IF VAR_mantisse2[2] >1 THEN
VAR_calcul_mantisse_temp.30:=TRUE;
VAR_mantisse2[2]:= VAR_mantisse2[2] -1;
ELSIF VAR_mantisse2[2] =1 THEN
VAR_calcul_mantisse_temp.30:=TRUE;
VAR_mantisse2[3]:=0;
VAR_mantisse2[4]:=0;
VAR_mantisse2[5]:=0;
VAR_mantisse2[6]:=0;
VAR_mantisse2[7]:=0;
VAR_mantisse2[8]:=0;
VAR_mantisse2[9]:=0;
VAR_mantisse2[10]:=0;
VAR_mantisse2[11]:=0;
VAR_mantisse2[12]:=0;
VAR_mantisse2[13]:=0;
VAR_mantisse2[14]:=0;
VAR_mantisse2[15]:=0;
VAR_mantisse2[16]:=0;
VAR_mantisse2[17]:=0;
VAR_mantisse2[18]:=0;
VAR_mantisse2[19]:=0;
VAR_mantisse2[20]:=0;
VAR_mantisse2[21]:=0;
VAR_mantisse2[22]:=0;
VAR_mantisse2[23]:=0;
VAR_mantisse2[24]:=0;
VAR_mantisse2[25]:=0;
VAR_mantisse2[26]:=0;
VAR_mantisse2[27]:=0;
VAR_mantisse2[28]:=0;
VAR_mantisse2[29]:=0;
VAR_mantisse2[30]:=0;
VAR_mantisse2[31]:=0;
VAR_mantisse2[32]:=0;
END_IF;

IF VAR_mantisse2[3] >1 THEN
VAR_calcul_mantisse_temp.29:=TRUE;
VAR_mantisse2[3]:= VAR_mantisse2[3] -1;
ELSIF VAR_mantisse2[3] =1 THEN
VAR_calcul_mantisse_temp.29:=TRUE;
VAR_mantisse2[4]:=0;
VAR_mantisse2[5]:=0;
VAR_mantisse2[6]:=0;
VAR_mantisse2[7]:=0;
VAR_mantisse2[8]:=0;
VAR_mantisse2[9]:=0;
VAR_mantisse2[10]:=0;
VAR_mantisse2[11]:=0;
VAR_mantisse2[12]:=0;
VAR_mantisse2[13]:=0;
VAR_mantisse2[14]:=0;
VAR_mantisse2[15]:=0;
VAR_mantisse2[16]:=0;
VAR_mantisse2[17]:=0;
VAR_mantisse2[18]:=0;
VAR_mantisse2[19]:=0;
VAR_mantisse2[20]:=0;
VAR_mantisse2[21]:=0;
VAR_mantisse2[22]:=0;
VAR_mantisse2[23]:=0;
VAR_mantisse2[24]:=0;
VAR_mantisse2[25]:=0;
VAR_mantisse2[26]:=0;
VAR_mantisse2[27]:=0;
VAR_mantisse2[28]:=0;
VAR_mantisse2[29]:=0;
VAR_mantisse2[30]:=0;
VAR_mantisse2[31]:=0;
VAR_mantisse2[32]:=0;
END_IF;

IF VAR_mantisse2[4] >1 THEN
VAR_calcul_mantisse_temp.28:=TRUE;
VAR_mantisse2[4]:= VAR_mantisse2[4] -1;
ELSIF VAR_mantisse2[4] =1 THEN
VAR_calcul_mantisse_temp.28:=TRUE;
VAR_mantisse2[5]:=0;
VAR_mantisse2[6]:=0;
VAR_mantisse2[7]:=0;
VAR_mantisse2[8]:=0;
VAR_mantisse2[9]:=0;
VAR_mantisse2[10]:=0;
VAR_mantisse2[11]:=0;
VAR_mantisse2[12]:=0;
VAR_mantisse2[13]:=0;
VAR_mantisse2[14]:=0;
VAR_mantisse2[15]:=0;
VAR_mantisse2[16]:=0;
VAR_mantisse2[17]:=0;
VAR_mantisse2[18]:=0;
VAR_mantisse2[19]:=0;
VAR_mantisse2[20]:=0;
VAR_mantisse2[21]:=0;
VAR_mantisse2[22]:=0;
VAR_mantisse2[23]:=0;
VAR_mantisse2[24]:=0;
VAR_mantisse2[25]:=0;
VAR_mantisse2[26]:=0;
VAR_mantisse2[27]:=0;
VAR_mantisse2[28]:=0;
VAR_mantisse2[29]:=0;
VAR_mantisse2[30]:=0;
VAR_mantisse2[31]:=0;
VAR_mantisse2[32]:=0;
END_IF;

IF VAR_mantisse2[5] >1 THEN
VAR_calcul_mantisse_temp.27:=TRUE;
VAR_mantisse2[5]:= VAR_mantisse2[5] -1;
ELSIF VAR_mantisse2[5] =1 THEN
VAR_calcul_mantisse_temp.27:=TRUE;
VAR_mantisse2[6]:=0;
VAR_mantisse2[7]:=0;
VAR_mantisse2[8]:=0;
VAR_mantisse2[9]:=0;
VAR_mantisse2[10]:=0;
VAR_mantisse2[11]:=0;
VAR_mantisse2[12]:=0;
VAR_mantisse2[13]:=0;
VAR_mantisse2[14]:=0;
VAR_mantisse2[15]:=0;
VAR_mantisse2[16]:=0;
VAR_mantisse2[17]:=0;
VAR_mantisse2[18]:=0;
VAR_mantisse2[19]:=0;
VAR_mantisse2[20]:=0;
VAR_mantisse2[21]:=0;
VAR_mantisse2[22]:=0;
VAR_mantisse2[23]:=0;
VAR_mantisse2[24]:=0;
VAR_mantisse2[25]:=0;
VAR_mantisse2[26]:=0;
VAR_mantisse2[27]:=0;
VAR_mantisse2[28]:=0;
VAR_mantisse2[29]:=0;
VAR_mantisse2[30]:=0;
VAR_mantisse2[31]:=0;
VAR_mantisse2[32]:=0;
END_IF;

IF VAR_mantisse2[6] >1 THEN
VAR_calcul_mantisse_temp.26:=TRUE;
VAR_mantisse2[6]:= VAR_mantisse2[6] -1;
ELSIF VAR_mantisse2[6] =1 THEN
VAR_calcul_mantisse_temp.26:=TRUE;
VAR_mantisse2[7]:=0;
VAR_mantisse2[8]:=0;
VAR_mantisse2[9]:=0;
VAR_mantisse2[10]:=0;
VAR_mantisse2[11]:=0;
VAR_mantisse2[12]:=0;
VAR_mantisse2[13]:=0;
VAR_mantisse2[14]:=0;
VAR_mantisse2[15]:=0;
VAR_mantisse2[16]:=0;
VAR_mantisse2[17]:=0;
VAR_mantisse2[18]:=0;
VAR_mantisse2[19]:=0;
VAR_mantisse2[20]:=0;
VAR_mantisse2[21]:=0;
VAR_mantisse2[22]:=0;
VAR_mantisse2[23]:=0;
VAR_mantisse2[24]:=0;
VAR_mantisse2[25]:=0;
VAR_mantisse2[26]:=0;
VAR_mantisse2[27]:=0;
VAR_mantisse2[28]:=0;
VAR_mantisse2[29]:=0;
VAR_mantisse2[30]:=0;
VAR_mantisse2[31]:=0;
VAR_mantisse2[32]:=0;
END_IF;

IF VAR_mantisse2[7] >1 THEN
VAR_calcul_mantisse_temp.25:=TRUE;
VAR_mantisse2[7]:= VAR_mantisse2[7] -1;
ELSIF VAR_mantisse2[7] =1 THEN
VAR_calcul_mantisse_temp.25:=TRUE;
VAR_mantisse2[8]:=0;
VAR_mantisse2[9]:=0;
VAR_mantisse2[10]:=0;
VAR_mantisse2[11]:=0;
VAR_mantisse2[12]:=0;
VAR_mantisse2[13]:=0;
VAR_mantisse2[14]:=0;
VAR_mantisse2[15]:=0;
VAR_mantisse2[16]:=0;
VAR_mantisse2[17]:=0;
VAR_mantisse2[18]:=0;
VAR_mantisse2[19]:=0;
VAR_mantisse2[20]:=0;
VAR_mantisse2[21]:=0;
VAR_mantisse2[22]:=0;
VAR_mantisse2[23]:=0;
VAR_mantisse2[24]:=0;
VAR_mantisse2[25]:=0;
VAR_mantisse2[26]:=0;
VAR_mantisse2[27]:=0;
VAR_mantisse2[28]:=0;
VAR_mantisse2[29]:=0;
VAR_mantisse2[30]:=0;
VAR_mantisse2[31]:=0;
VAR_mantisse2[32]:=0;
END_IF;

IF VAR_mantisse2[8] >1 THEN
VAR_calcul_mantisse_temp.24:=TRUE;
VAR_mantisse2[8]:= VAR_mantisse2[8] -1;
ELSIF VAR_mantisse2[8] =1 THEN
VAR_calcul_mantisse_temp.24:=TRUE;
VAR_mantisse2[9]:=0;
VAR_mantisse2[10]:=0;
VAR_mantisse2[11]:=0;
VAR_mantisse2[12]:=0;
VAR_mantisse2[13]:=0;
VAR_mantisse2[14]:=0;
VAR_mantisse2[15]:=0;
VAR_mantisse2[16]:=0;
VAR_mantisse2[17]:=0;
VAR_mantisse2[18]:=0;
VAR_mantisse2[19]:=0;
VAR_mantisse2[20]:=0;
VAR_mantisse2[21]:=0;
VAR_mantisse2[22]:=0;
VAR_mantisse2[23]:=0;
VAR_mantisse2[24]:=0;
VAR_mantisse2[25]:=0;
VAR_mantisse2[26]:=0;
VAR_mantisse2[27]:=0;
VAR_mantisse2[28]:=0;
VAR_mantisse2[29]:=0;
VAR_mantisse2[30]:=0;
VAR_mantisse2[31]:=0;
VAR_mantisse2[32]:=0;
END_IF;

IF VAR_mantisse2[9] >1 THEN
VAR_calcul_mantisse_temp.23:=TRUE;
VAR_mantisse2[9]:= VAR_mantisse2[9] -1;
ELSIF VAR_mantisse2[9] =1 THEN
VAR_calcul_mantisse_temp.23:=TRUE;
VAR_mantisse2[10]:=0;
VAR_mantisse2[11]:=0;
VAR_mantisse2[12]:=0;
VAR_mantisse2[13]:=0;
VAR_mantisse2[14]:=0;
VAR_mantisse2[15]:=0;
VAR_mantisse2[16]:=0;
VAR_mantisse2[17]:=0;
VAR_mantisse2[18]:=0;
VAR_mantisse2[19]:=0;
VAR_mantisse2[20]:=0;
VAR_mantisse2[21]:=0;
VAR_mantisse2[22]:=0;
VAR_mantisse2[23]:=0;
VAR_mantisse2[24]:=0;
VAR_mantisse2[25]:=0;
VAR_mantisse2[26]:=0;
VAR_mantisse2[27]:=0;
VAR_mantisse2[28]:=0;
VAR_mantisse2[29]:=0;
VAR_mantisse2[30]:=0;
VAR_mantisse2[31]:=0;
VAR_mantisse2[32]:=0;
END_IF;

IF VAR_mantisse2[10] >1 THEN
VAR_calcul_mantisse_temp.22:=TRUE;
VAR_mantisse2[10]:= VAR_mantisse2[10] -1;
ELSIF VAR_mantisse2[10] =1 THEN
VAR_calcul_mantisse_temp.22:=TRUE;
VAR_mantisse2[11]:=0;
VAR_mantisse2[12]:=0;
VAR_mantisse2[13]:=0;
VAR_mantisse2[14]:=0;
VAR_mantisse2[15]:=0;
VAR_mantisse2[16]:=0;
VAR_mantisse2[17]:=0;
VAR_mantisse2[18]:=0;
VAR_mantisse2[19]:=0;
VAR_mantisse2[20]:=0;
VAR_mantisse2[21]:=0;
VAR_mantisse2[22]:=0;
VAR_mantisse2[23]:=0;
VAR_mantisse2[24]:=0;
VAR_mantisse2[25]:=0;
VAR_mantisse2[26]:=0;
VAR_mantisse2[27]:=0;
VAR_mantisse2[28]:=0;
VAR_mantisse2[29]:=0;
VAR_mantisse2[30]:=0;
VAR_mantisse2[31]:=0;
VAR_mantisse2[32]:=0;
END_IF;
IF VAR_mantisse2[11] >1 THEN
VAR_calcul_mantisse_temp.21:=TRUE;
VAR_mantisse2[11]:= VAR_mantisse2[11] -1;
ELSIF VAR_mantisse2[11] =1 THEN
VAR_calcul_mantisse_temp.21:=TRUE;
VAR_mantisse2[12]:=0;
VAR_mantisse2[13]:=0;
VAR_mantisse2[14]:=0;
VAR_mantisse2[15]:=0;
VAR_mantisse2[16]:=0;
VAR_mantisse2[17]:=0;
VAR_mantisse2[18]:=0;
VAR_mantisse2[19]:=0;
VAR_mantisse2[20]:=0;
VAR_mantisse2[21]:=0;
VAR_mantisse2[22]:=0;
VAR_mantisse2[23]:=0;
VAR_mantisse2[24]:=0;
VAR_mantisse2[25]:=0;
VAR_mantisse2[26]:=0;
VAR_mantisse2[27]:=0;
VAR_mantisse2[28]:=0;
VAR_mantisse2[29]:=0;
VAR_mantisse2[30]:=0;
VAR_mantisse2[31]:=0;
VAR_mantisse2[32]:=0;
END_IF;
IF VAR_mantisse2[12] >1 THEN
VAR_calcul_mantisse_temp.20:=TRUE;
VAR_mantisse2[12]:= VAR_mantisse2[12] -1;
ELSIF VAR_mantisse2[12] =1 THEN
VAR_calcul_mantisse_temp.20:=TRUE;
VAR_mantisse2[13]:=0;
VAR_mantisse2[14]:=0;
VAR_mantisse2[15]:=0;
VAR_mantisse2[16]:=0;
VAR_mantisse2[17]:=0;
VAR_mantisse2[18]:=0;
VAR_mantisse2[19]:=0;
VAR_mantisse2[20]:=0;
VAR_mantisse2[21]:=0;
VAR_mantisse2[22]:=0;
VAR_mantisse2[23]:=0;
VAR_mantisse2[24]:=0;
VAR_mantisse2[25]:=0;
VAR_mantisse2[26]:=0;
VAR_mantisse2[27]:=0;
VAR_mantisse2[28]:=0;
VAR_mantisse2[29]:=0;
VAR_mantisse2[30]:=0;
VAR_mantisse2[31]:=0;
VAR_mantisse2[32]:=0;
END_IF;
IF VAR_mantisse2[13] >1 THEN
VAR_calcul_mantisse_temp.19:=TRUE;
VAR_mantisse2[13]:= VAR_mantisse2[13] -1;
ELSIF VAR_mantisse2[13] =1 THEN
VAR_calcul_mantisse_temp.19:=TRUE;
VAR_mantisse2[14]:=0;
VAR_mantisse2[15]:=0;
VAR_mantisse2[16]:=0;
VAR_mantisse2[17]:=0;
VAR_mantisse2[18]:=0;
VAR_mantisse2[19]:=0;
VAR_mantisse2[20]:=0;
VAR_mantisse2[21]:=0;
VAR_mantisse2[22]:=0;
VAR_mantisse2[23]:=0;
VAR_mantisse2[24]:=0;
VAR_mantisse2[25]:=0;
VAR_mantisse2[26]:=0;
VAR_mantisse2[27]:=0;
VAR_mantisse2[28]:=0;
VAR_mantisse2[29]:=0;
VAR_mantisse2[30]:=0;
VAR_mantisse2[31]:=0;
VAR_mantisse2[32]:=0;
END_IF;
IF VAR_mantisse2[14] >1 THEN
VAR_calcul_mantisse_temp.18:=TRUE;
VAR_mantisse2[14]:= VAR_mantisse2[14] -1;
ELSIF VAR_mantisse2[14] =1 THEN
VAR_calcul_mantisse_temp.18:=TRUE;
VAR_mantisse2[15]:=0;
VAR_mantisse2[16]:=0;
VAR_mantisse2[17]:=0;
VAR_mantisse2[18]:=0;
VAR_mantisse2[19]:=0;
VAR_mantisse2[20]:=0;
VAR_mantisse2[21]:=0;
VAR_mantisse2[22]:=0;
VAR_mantisse2[23]:=0;
VAR_mantisse2[24]:=0;
VAR_mantisse2[25]:=0;
VAR_mantisse2[26]:=0;
VAR_mantisse2[27]:=0;
VAR_mantisse2[28]:=0;
VAR_mantisse2[29]:=0;
VAR_mantisse2[30]:=0;
VAR_mantisse2[31]:=0;
VAR_mantisse2[32]:=0;
END_IF;

IF VAR_mantisse2[15] >1 THEN
VAR_calcul_mantisse_temp.17:=TRUE;
VAR_mantisse2[15]:= VAR_mantisse2[15] -1;
ELSIF VAR_mantisse2[15] =1 THEN
VAR_calcul_mantisse_temp.17:=TRUE;
VAR_mantisse2[16]:=0;
VAR_mantisse2[17]:=0;
VAR_mantisse2[18]:=0;
VAR_mantisse2[19]:=0;
VAR_mantisse2[20]:=0;
VAR_mantisse2[21]:=0;
VAR_mantisse2[22]:=0;
VAR_mantisse2[23]:=0;
VAR_mantisse2[24]:=0;
VAR_mantisse2[25]:=0;
VAR_mantisse2[26]:=0;
VAR_mantisse2[27]:=0;
VAR_mantisse2[28]:=0;
VAR_mantisse2[29]:=0;
VAR_mantisse2[30]:=0;
VAR_mantisse2[31]:=0;
VAR_mantisse2[32]:=0;
END_IF;
IF VAR_mantisse2[16] >1 THEN
VAR_calcul_mantisse_temp.16:=TRUE;
VAR_mantisse2[16]:= VAR_mantisse2[16] -1;
ELSIF VAR_mantisse2[16] =1 THEN
VAR_calcul_mantisse_temp.16:=TRUE;
VAR_mantisse2[17]:=0;
VAR_mantisse2[18]:=0;
VAR_mantisse2[19]:=0;
VAR_mantisse2[20]:=0;
VAR_mantisse2[21]:=0;
VAR_mantisse2[22]:=0;
VAR_mantisse2[23]:=0;
VAR_mantisse2[24]:=0;
VAR_mantisse2[25]:=0;
VAR_mantisse2[26]:=0;
VAR_mantisse2[27]:=0;
VAR_mantisse2[28]:=0;
VAR_mantisse2[29]:=0;
VAR_mantisse2[30]:=0;
VAR_mantisse2[31]:=0;
VAR_mantisse2[32]:=0;
END_IF;
IF VAR_mantisse2[17] >1 THEN
VAR_calcul_mantisse_temp.15:=TRUE;
VAR_mantisse2[17]:= VAR_mantisse2[17] -1;
ELSIF VAR_mantisse2[17] =1 THEN
VAR_calcul_mantisse_temp.15:=TRUE;
VAR_mantisse2[18]:=0;
VAR_mantisse2[19]:=0;
VAR_mantisse2[20]:=0;
VAR_mantisse2[21]:=0;
VAR_mantisse2[22]:=0;
VAR_mantisse2[23]:=0;
VAR_mantisse2[24]:=0;
VAR_mantisse2[25]:=0;
VAR_mantisse2[26]:=0;
VAR_mantisse2[27]:=0;
VAR_mantisse2[28]:=0;
VAR_mantisse2[29]:=0;
VAR_mantisse2[30]:=0;
VAR_mantisse2[31]:=0;
VAR_mantisse2[32]:=0;
END_IF;
IF VAR_mantisse2[18] >1 THEN
VAR_calcul_mantisse_temp.14:=TRUE;
VAR_mantisse2[18]:= VAR_mantisse2[18] -1;
ELSIF VAR_mantisse2[18] =1 THEN
VAR_calcul_mantisse_temp.14:=TRUE;
VAR_mantisse2[19]:=0;
VAR_mantisse2[20]:=0;
VAR_mantisse2[21]:=0;
VAR_mantisse2[22]:=0;
VAR_mantisse2[23]:=0;
VAR_mantisse2[24]:=0;
VAR_mantisse2[25]:=0;
VAR_mantisse2[26]:=0;
VAR_mantisse2[27]:=0;
VAR_mantisse2[28]:=0;
VAR_mantisse2[29]:=0;
VAR_mantisse2[30]:=0;
VAR_mantisse2[31]:=0;
VAR_mantisse2[32]:=0;
END_IF;
IF VAR_mantisse2[19] >1 THEN
VAR_calcul_mantisse_temp.13:=TRUE;
VAR_mantisse2[19]:= VAR_mantisse2[19] -1;
ELSIF VAR_mantisse2[19] =1 THEN
VAR_calcul_mantisse_temp.13:=TRUE;
VAR_mantisse2[20]:=0;
VAR_mantisse2[21]:=0;
VAR_mantisse2[22]:=0;
VAR_mantisse2[23]:=0;
VAR_mantisse2[24]:=0;
VAR_mantisse2[25]:=0;
VAR_mantisse2[26]:=0;
VAR_mantisse2[27]:=0;
VAR_mantisse2[28]:=0;
VAR_mantisse2[29]:=0;
VAR_mantisse2[30]:=0;
VAR_mantisse2[31]:=0;
VAR_mantisse2[32]:=0;
END_IF;
IF VAR_mantisse2[20] >1 THEN
VAR_calcul_mantisse_temp.12:=TRUE;
VAR_mantisse2[20]:= VAR_mantisse2[20] -1;
ELSIF VAR_mantisse2[20] =1 THEN
VAR_calcul_mantisse_temp.12:=TRUE;
VAR_mantisse2[21]:=0;
VAR_mantisse2[22]:=0;
VAR_mantisse2[23]:=0;
VAR_mantisse2[24]:=0;
VAR_mantisse2[25]:=0;
VAR_mantisse2[26]:=0;
VAR_mantisse2[27]:=0;
VAR_mantisse2[28]:=0;
VAR_mantisse2[29]:=0;
VAR_mantisse2[30]:=0;
VAR_mantisse2[31]:=0;
VAR_mantisse2[32]:=0;
END_IF;
IF VAR_mantisse2[21] >1 THEN
VAR_calcul_mantisse_temp.11:=TRUE;
VAR_mantisse2[21]:= VAR_mantisse2[21] -1;
ELSIF VAR_mantisse2[21] =1 THEN
VAR_calcul_mantisse_temp.11:=TRUE;
VAR_mantisse2[22]:=0;
VAR_mantisse2[23]:=0;
VAR_mantisse2[24]:=0;
VAR_mantisse2[25]:=0;
VAR_mantisse2[26]:=0;
VAR_mantisse2[27]:=0;
VAR_mantisse2[28]:=0;
VAR_mantisse2[29]:=0;
VAR_mantisse2[30]:=0;
VAR_mantisse2[31]:=0;
VAR_mantisse2[32]:=0;
END_IF;
IF VAR_mantisse2[22] >1 THEN
VAR_calcul_mantisse_temp.10:=TRUE;
VAR_mantisse2[22]:= VAR_mantisse2[22] -1;
ELSIF VAR_mantisse2[22] =1 THEN
VAR_calcul_mantisse_temp.10:=TRUE;
VAR_mantisse2[23]:=0;
VAR_mantisse2[24]:=0;
VAR_mantisse2[25]:=0;
VAR_mantisse2[26]:=0;
VAR_mantisse2[27]:=0;
VAR_mantisse2[28]:=0;
VAR_mantisse2[29]:=0;
VAR_mantisse2[30]:=0;
VAR_mantisse2[31]:=0;
VAR_mantisse2[32]:=0;
END_IF;
IF VAR_mantisse2[23] >1 THEN
VAR_calcul_mantisse_temp.9:=TRUE;
VAR_mantisse2[23]:= VAR_mantisse2[23] -1;
ELSIF VAR_mantisse2[23] =1 THEN
VAR_calcul_mantisse_temp.9:=TRUE;
VAR_mantisse2[24]:=0;
VAR_mantisse2[25]:=0;
VAR_mantisse2[26]:=0;
VAR_mantisse2[27]:=0;
VAR_mantisse2[28]:=0;
VAR_mantisse2[29]:=0;
VAR_mantisse2[30]:=0;
VAR_mantisse2[31]:=0;
VAR_mantisse2[32]:=0;
END_IF;
IF VAR_mantisse2[24] >1 THEN
VAR_calcul_mantisse_temp.8:=TRUE;
VAR_mantisse2[24]:= VAR_mantisse2[24] -1;
ELSIF VAR_mantisse2[24] =1 THEN
VAR_calcul_mantisse_temp.8:=TRUE;
VAR_mantisse2[25]:=0;
VAR_mantisse2[26]:=0;
VAR_mantisse2[27]:=0;
VAR_mantisse2[28]:=0;
VAR_mantisse2[29]:=0;
VAR_mantisse2[30]:=0;
VAR_mantisse2[31]:=0;
VAR_mantisse2[32]:=0;
END_IF;
IF VAR_mantisse2[25] >1 THEN
VAR_calcul_mantisse_temp.7:=TRUE;
VAR_mantisse2[25]:= VAR_mantisse2[25] -1;
ELSIF VAR_mantisse2[25] =1 THEN
VAR_calcul_mantisse_temp.7:=TRUE;
VAR_mantisse2[26]:=0;
VAR_mantisse2[27]:=0;
VAR_mantisse2[28]:=0;
VAR_mantisse2[29]:=0;
VAR_mantisse2[30]:=0;
VAR_mantisse2[31]:=0;
VAR_mantisse2[32]:=0;
END_IF;
IF VAR_mantisse2[26] >1 THEN
VAR_calcul_mantisse_temp.6:=TRUE;
VAR_mantisse2[26]:= VAR_mantisse2[26] -1;
ELSIF VAR_mantisse2[26] =1 THEN
VAR_calcul_mantisse_temp.6:=TRUE;
VAR_mantisse2[27]:=0;
VAR_mantisse2[28]:=0;
VAR_mantisse2[29]:=0;
VAR_mantisse2[30]:=0;
VAR_mantisse2[31]:=0;
VAR_mantisse2[32]:=0;
END_IF;
IF VAR_mantisse2[27] >1 THEN
VAR_calcul_mantisse_temp.5:=TRUE;
VAR_mantisse2[27]:= VAR_mantisse2[27] -1;
ELSIF VAR_mantisse2[27] =1 THEN
VAR_calcul_mantisse_temp.5:=TRUE;
VAR_mantisse2[28]:=0;
VAR_mantisse2[29]:=0;
VAR_mantisse2[30]:=0;
VAR_mantisse2[31]:=0;
VAR_mantisse2[32]:=0;
END_IF;
IF VAR_mantisse2[28] >1 THEN
VAR_calcul_mantisse_temp.4:=TRUE;
VAR_mantisse2[28]:= VAR_mantisse2[28] -1;
ELSIF VAR_mantisse2[28] =1 THEN
VAR_calcul_mantisse_temp.4:=TRUE;
VAR_mantisse2[29]:=0;
VAR_mantisse2[30]:=0;
VAR_mantisse2[31]:=0;
VAR_mantisse2[32]:=0;
END_IF;
IF VAR_mantisse2[29] >1 THEN
VAR_calcul_mantisse_temp.3:=TRUE;
VAR_mantisse2[29]:= VAR_mantisse2[29] -1;
ELSIF VAR_mantisse2[29] =1 THEN
VAR_calcul_mantisse_temp.3:=TRUE;
VAR_mantisse2[30]:=0;
VAR_mantisse2[31]:=0;
VAR_mantisse2[32]:=0;
END_IF;
IF VAR_mantisse2[30] >1 THEN
VAR_calcul_mantisse_temp.2:=TRUE;
VAR_mantisse2[30]:= VAR_mantisse2[30] -1;
ELSIF VAR_mantisse2[30] =1 THEN
VAR_calcul_mantisse_temp.2:=TRUE;
VAR_mantisse2[31]:=0;
VAR_mantisse2[32]:=0;
END_IF;
IF VAR_mantisse2[31] >1 THEN
VAR_calcul_mantisse_temp.1:=TRUE;
VAR_mantisse2[31]:= VAR_mantisse2[31] -1;
ELSIF VAR_mantisse2[31] =1 THEN
VAR_calcul_mantisse_temp.1:=TRUE;
VAR_mantisse2[32]:=0;
END_IF;
IF VAR_mantisse2[32] >1 THEN
VAR_calcul_mantisse_temp.0:=TRUE;
VAR_mantisse2[32]:= VAR_mantisse2[32] -1;
ELSIF VAR_mantisse2[32] =1 THEN
VAR_calcul_mantisse_temp.0:=TRUE;
END_IF;
END_FOR

VAR_calcul_mantisse_temp2:=VAR_calcul_mantisse_temp;
VAR_value2:=VAR_value_entiere_corrige;
N:=0;
FOR I:=1 TO 32 DO

IF VAR_mantisse2[I] = 1 THEN
	N:=INT_TO_BYTE(I);
END_IF
END_FOR

Var_decalage_bit:=32-N;
VAR_mantisse_decimal:=ROR(VAR_calcul_mantisse_temp2,Var_decalage_bit);
VAR_mantisse_entier:=ROL(VAR_value2,N);

VAR_mantisse_final:= VAR_mantisse_entier OR VAR_mantisse_decimal;

IF VAR_mantisse_final.31=TRUE THEN
VAR_nb_zero:=0;
ELSIF VAR_mantisse_final.30=TRUE THEN
VAR_nb_zero:=1;
ELSIF VAR_mantisse_final.29=TRUE THEN
VAR_nb_zero:=2;
ELSIF VAR_mantisse_final.28=TRUE THEN
VAR_nb_zero:=3;
ELSIF VAR_mantisse_final.27=TRUE THEN
VAR_nb_zero:=4;
ELSIF VAR_mantisse_final.26=TRUE THEN
VAR_nb_zero:=5;
ELSIF VAR_mantisse_final.25=TRUE THEN
VAR_nb_zero:=6;
ELSIF VAR_mantisse_final.24=TRUE THEN
VAR_nb_zero:=7;
ELSIF VAR_mantisse_final.23=TRUE THEN
VAR_nb_zero:=8;
ELSIF VAR_mantisse_final.22=TRUE THEN
VAR_nb_zero:=9;
ELSIF VAR_mantisse_final.21=TRUE THEN
VAR_nb_zero:=10;
ELSIF VAR_mantisse_final.20=TRUE THEN
VAR_nb_zero:=11;
ELSIF VAR_mantisse_final.19=TRUE THEN
VAR_nb_zero:=12;
ELSIF VAR_mantisse_final.18=TRUE THEN
VAR_nb_zero:=13;
ELSIF VAR_mantisse_final.17=TRUE THEN
VAR_nb_zero:=14;
ELSIF VAR_mantisse_final.16=TRUE THEN
VAR_nb_zero:=15;
ELSIF VAR_mantisse_final.15=TRUE THEN
VAR_nb_zero:=16;
ELSIF VAR_mantisse_final.14=TRUE THEN
VAR_nb_zero:=17;
ELSIF VAR_mantisse_final.13=TRUE THEN
VAR_nb_zero:=18;
ELSIF VAR_mantisse_final.12=TRUE THEN
VAR_nb_zero:=19;
ELSIF VAR_mantisse_final.11=TRUE THEN
VAR_nb_zero:=20;
ELSIF VAR_mantisse_final.10=TRUE THEN
VAR_nb_zero:=21;
ELSIF VAR_mantisse_final.9=TRUE THEN
VAR_nb_zero:=22;
ELSIF VAR_mantisse_final.8=TRUE THEN
VAR_nb_zero:=23;
ELSIF VAR_mantisse_final.7=TRUE THEN
VAR_nb_zero:=24;
ELSIF VAR_mantisse_final.6=TRUE THEN
VAR_nb_zero:=25;
ELSIF VAR_mantisse_final.5=TRUE THEN
VAR_nb_zero:=26;
ELSIF VAR_mantisse_final.4=TRUE THEN
VAR_nb_zero:=27;
ELSIF VAR_mantisse_final.3=TRUE THEN
VAR_nb_zero:=28;
ELSIF VAR_mantisse_final.2=TRUE THEN
VAR_nb_zero:=29;
ELSIF VAR_mantisse_final.1=TRUE THEN
VAR_nb_zero:=30;
ELSIF VAR_mantisse_final.0=TRUE THEN
VAR_nb_zero:=31;
END_IF

 VAR_calcul_exposant := (32 - VAR_nb_zero - N - 1) + 127;

J:=INT_TO_BYTE(VAR_nb_zero);

VAR_mantisse_final2:=ROL(VAR_mantisse_final ,J);

VAR_calcul_sortie.31 := VAR_signe;

VAR_calcul_sortie.30 := VAR_calcul_exposant.7;
VAR_calcul_sortie.29 := VAR_calcul_exposant.6;
VAR_calcul_sortie.28 := VAR_calcul_exposant.5;
VAR_calcul_sortie.27 := VAR_calcul_exposant.4 ;
VAR_calcul_sortie.26 := VAR_calcul_exposant.3;
VAR_calcul_sortie.25 := VAR_calcul_exposant.2;
VAR_calcul_sortie.24 := VAR_calcul_exposant.1 ;
VAR_calcul_sortie.23 := VAR_calcul_exposant.0;

VAR_calcul_sortie.22 := VAR_mantisse_final2.30;
VAR_calcul_sortie.21 := VAR_mantisse_final2.29;
VAR_calcul_sortie.20 := VAR_mantisse_final2.28;
VAR_calcul_sortie.19 := VAR_mantisse_final2.27;
VAR_calcul_sortie.18 := VAR_mantisse_final2.26;
VAR_calcul_sortie.17 := VAR_mantisse_final2.25;
VAR_calcul_sortie.16 := VAR_mantisse_final2.24;
VAR_calcul_sortie.15 := VAR_mantisse_final2.23;
VAR_calcul_sortie.14 := VAR_mantisse_final2.22;
VAR_calcul_sortie.13 := VAR_mantisse_final2.21;
VAR_calcul_sortie.12 := VAR_mantisse_final2.20;
VAR_calcul_sortie.11 := VAR_mantisse_final2.19;
VAR_calcul_sortie.10 := VAR_mantisse_final2.18;
VAR_calcul_sortie.9 := VAR_mantisse_final2.17;
VAR_calcul_sortie.8 := VAR_mantisse_final2.16;
VAR_calcul_sortie.7 := VAR_mantisse_final2.15;
VAR_calcul_sortie.6 := VAR_mantisse_final2.14;
VAR_calcul_sortie.5 := VAR_mantisse_final2.13;
VAR_calcul_sortie.4 := VAR_mantisse_final2.12;
VAR_calcul_sortie.3 := VAR_mantisse_final2.11;
VAR_calcul_sortie.2 := VAR_mantisse_final2.10;
VAR_calcul_sortie.1 := VAR_mantisse_final2.9;
VAR_calcul_sortie.0 := VAR_mantisse_final2.8;

OUTPUT[0].0 := VAR_calcul_sortie.0;
OUTPUT[0].1 := VAR_calcul_sortie.1;
OUTPUT[0].2 := VAR_calcul_sortie.2;
OUTPUT[0].3 := VAR_calcul_sortie.3;
OUTPUT[0].4 := VAR_calcul_sortie.4;
OUTPUT[0].5 := VAR_calcul_sortie.5;
OUTPUT[0].6 := VAR_calcul_sortie.6;
OUTPUT[0].7 := VAR_calcul_sortie.7;

OUTPUT[1].0 := VAR_calcul_sortie.8;
OUTPUT[1].1 := VAR_calcul_sortie.9;
OUTPUT[1].2 := VAR_calcul_sortie.10;
OUTPUT[1].3 := VAR_calcul_sortie.11;
OUTPUT[1].4 := VAR_calcul_sortie.12;
OUTPUT[1].5 := VAR_calcul_sortie.13;
OUTPUT[1].6 := VAR_calcul_sortie.14;
OUTPUT[1].7 := VAR_calcul_sortie.15;

OUTPUT[2].0 := VAR_calcul_sortie.16;
OUTPUT[2].1 := VAR_calcul_sortie.17;
OUTPUT[2].2 := VAR_calcul_sortie.18;
OUTPUT[2].3 := VAR_calcul_sortie.19;
OUTPUT[2].4 := VAR_calcul_sortie.20;
OUTPUT[2].5 := VAR_calcul_sortie.21;
OUTPUT[2].6 := VAR_calcul_sortie.22;
OUTPUT[2].7 := VAR_calcul_sortie.23;

OUTPUT[3].0 := VAR_calcul_sortie.24;
OUTPUT[3].1 := VAR_calcul_sortie.25;
OUTPUT[3].2 := VAR_calcul_sortie.26;
OUTPUT[3].3 := VAR_calcul_sortie.27;
OUTPUT[3].4 := VAR_calcul_sortie.28;
OUTPUT[3].5 := VAR_calcul_sortie.29;
OUTPUT[3].6 := VAR_calcul_sortie.30;
OUTPUT[3].7 := VAR_calcul_sortie.31;

END_FUNCTION_BLOCK

// ---- POUs/Fonction/ETHER COM/BLOCK_XTC_CLIENT_EXCHANGE.TcPOU
FUNCTION_BLOCK BLOCK_XTC_CLIENT_EXCHANGE
(* Fonction de lecture / écriture sur port TcpIP*)
(* version 0 - SP - 24/02/2015*)


VAR_INPUT
	hSocket				: T_HSOCKET;	(*socket*)
	TxBuffer				: ARRAY[0..MAX_TXBUFFER_SIZE] OF BYTE;
	bExecute			: BOOL;			(*bit de déclenchelent de l'émission/réception - sur front montant*)
	nbExpectedChar		: UDINT;			(*nombre de caractère attendu en réception*)
	nbTransmittedChar	: UDINT;			(*nombre de caractère transmis à l'émission*)
	PRM_RECEIVE_POLLING_TIME		 		: TIME := T#1s;	(*temporisation de polling de réception*)
	PRM_RECEIVE_TIMEOUT						: TIME := T#10s;	(*temporisation de timeout de communication*)

END_VAR
VAR_OUTPUT
	bBusy 				: BOOL;			(*processus d'emission/réception occupé*)
	bError				: BOOL;			(*processus d'emission/réception en erreur*)
	nErrId				: UDINT;			(*n° d'erreur*)
	nstepInError			: UDINT;			(*n° d'étape sur laquelle s'est produite l'erreur*)
	ErrDescription		: T_MaxString;	(*chaine de caractère d'intitulé de l'erreur*)
	rxBuffer				: ARRAY[0..MAX_RXBUFFER_SIZE] OF BYTE; (*réponse du serveur en mode buffer*)
	STATE_Com_Err_Counter:	UDINT;
	STATE_nbReceptedChar:	UDINT;			(*nombre effectif de caractère recu - peut différer du nombre de caractère attendu dans le cas d'une trame
										d'erreur*)

END_VAR
VAR
	fbSocketSend		: FB_SocketSend := ( sSrvNetID := '', tTimeout := DEFAULT_ADS_TIMEOUT );
	fbSocketReceive		: FB_SocketReceive := ( sSrvNetID := '', tTimeout := DEFAULT_ADS_TIMEOUT );
	fbReceiveTON		: TON;		(*tempo pour polling de réception*)
	fbDisconnectTON		: TON;		(*tempo de time out*)
	RisingEdge			: R_TRIG;
	eStep				: E_DataExchaSteps;
	cbReceived, startPos, endPos, idx	: UDINT;
	cbFrame				: UDINT;
	Temp_rxBuffer		: ARRAY[0..MAX_RXBUFFER_SIZE] OF BYTE;
	I					: INT; 		(*Compteur d'itération*)
	LOG_COM			: ARRAY[0..MAX_BUFFER_DIALOG] OF STRUCT_LOG_TCPIP_CLIENT;	(*buffer de chaine en émission*)
	VAR_COUNT_RETRY:	INT;		(*Compteur de tentative de retransmission du paramètre*)
END_VAR
VAR_TEMP
	Temp_byte:			BYTE;
END_VAR

RisingEdge( CLK := bExecute );	(*gestion du front montant de la demande d'exécution*)
CASE eStep OF

	DATAEXCHA_STATE_IDLE:	(*etape 0 - fonction d'émisson réception à l'arrêt*)
		IF RisingEdge.Q THEN		(*demande d'emission/réception sur FM du bit bexecute*)
		VAR_COUNT_RETRY := 0;
			(*RAZ du buffer de réception et du buffer de réception temporaire*)
			FOR i:=0 TO UDINT_TO_INT(MAX_RXBUFFER_SIZE) DO
				Temp_RxBuffer[i] := 0;
				RxBuffer[i] :=0;
			END_FOR
			bBusy := TRUE;							(*processus d'émission / réception occupé*)
			bError := FALSE;							(* RAZ drapeau d'erreur*)
			nErrid := 0;								(*RAZ du type d'érreur*)
			fbReceiveTON( IN := FALSE, PT := T#0s ); 	(* Réglage du buffer de réception à 0 pour lire asap *)
			fbDisconnectTON( IN := FALSE, PT := T#0s );	(* désactivation du timer de timeout *)
			eStep := DATAEXCHA_STATE_SEND_START;
		END_IF

	DATAEXCHA_STATE_SEND_START:		(*Etape 1 -  Envoi de la trame au serveur*)
		fbSocketSend( bExecute := FALSE );
		CbReceived := 0;
		(*on envoie le buffer d'émission*)
		fbSocketSend(
					hSocket	:= hSocket,
					pSrc	:= ADR(TxBuffer),
					cblen 	:= NbTransmittedChar, (* longueur de chaine sans le délimiteur *)
					bExecute:= TRUE,
					);
		fbsocketSend.cblen := NbTransmittedChar; (*longueur de chaine à envoyer*)

		SHIFT_BUFFER_DIALOG(); (*décalage du buffer de mémoire des dernières trames d'émission*)

		(*mémorisation du buffer d'émission dans le journal des échanges *)
		 MEMCPY( ADR(LOG_COM[0].TX),ADR(TxBuffer),FbSocketSend.Cblen);

		eStep := DATAEXCHA_STATE_SEND_WAIT;

	DATAEXCHA_STATE_SEND_WAIT:			(* Etape 2 - attente de la fin de l'envoi de la trame*)
		fbSocketSend( bExecute := FALSE );
		IF NOT fbSocketSend.bBusy THEN	(*si fin de l'emission*)
			IF NOT fbSocketSend.bError THEN	(*pas d'erreur*)
				eStep := DATAEXCHA_STATE_RECEIVE_START;
			ELSE	(*detection d'une erreur d'émission*)
				(*LogError( 'FB_SocketSend (local client)', fbSocketSend.nErrId );*)
				nErrId := fbSocketSend.nErrId;
				nstepInError := 2;
				ErrDescription := CONCAT('FB_ClientDataExcha - SENDING ERROR: ', UDINT_TO_STRING(nErrId));
				LOG_COM[0].ERR := ErrDescription;
				eStep := DATAEXCHA_STATE_ERROR;
			END_IF
		END_IF

	DATAEXCHA_STATE_RECEIVE_START: 	(*Etape 3 - gestion de la réception*)
		fbDisconnectTON(  );	(*lancement de la tempo de timeout : desactivée au premier appel*)
		fbReceiveTON( IN := TRUE );	(*temporisation de polling de reception - lancé avec délai 0ms au premier appel*)
		IF fbReceiveTON.Q THEN
			fbReceiveTON( IN := FALSE );
			fbSocketReceive( bExecute := FALSE );
			fbSocketReceive(  hSocket:= hSocket,
							pDest:= ADR( Temp_rxBuffer ) + cbReceived,	(*ajouté au buffer de réception à partir du dernier index CbReceived*)
							cbLen:= SIZEOF( Temp_rxBuffer ) - cbReceived,   (*longueur max = longeur du buffer - dernier index CbReceived*)
							bExecute:= TRUE );
			eStep := DATAEXCHA_STATE_RECEIVE_WAIT;
		END_IF

	DATAEXCHA_STATE_RECEIVE_WAIT:			(*étape 4 - attente de la fin de réception*)
		fbSocketReceive( bExecute := FALSE );
		IF NOT fbSocketReceive.bBusy THEN		(*si pas fonction de réception en cours*)
			IF NOT fbSocketReceive.bError THEN	(*si pas d'erreur*)
				(*et si des bytes ont été reçu*)
				IF (fbSocketReceive.nRecBytes > 0) THEN(* si on a reçu des informations *)
					startPos 		:= cbReceived;(* calcul de l'index de début de la nouvelle trame lue dans le buffer *)
					endPos  		:= cbReceived + fbSocketReceive.nRecBytes  - 1;(* calcul de l'index de fin de la nouvelle trame lue dans le buffer *)
					cbReceived 	:= cbReceived + fbSocketReceive.nRecBytes;(* recalcule le nombre total de caractères reçus depuis la requête en émission*)
					cbFrame		:= 0;(* remise à 0 de la  *)

					IF  (cbReceived < MAX_RXBUFFER_SIZE) (* contrôle de débordement *)  THEN

						fbReceiveTON( PT := T#0s ); (* bytes reçus =>on fixe la pariode de pooling a 0ms *)
						fbDisconnectTON( IN := FALSE );(* bytes recus => on ihnibe la tempo de timeout *)

						(*analyse des 2 premiers octets de la trame*)
						IF (cbReceived >=3)  THEN
							(*reception d'un message d'erreur de l'XTC*)
							IF ((temp_RxBuffer[0] + (Temp_RxBuffer[1] * 256)) = 6) AND (Temp_RxBuffer[2] = 16#80) THEN
								nbExpectedChar:= 6;	(*on corrige le nombre de caractère attendu*)
								STATE_nbReceptedChar:=6;
							END_IF
							(*Reception d'un message au format erroné - mauvais caractère CCB*)
							IF NOT (Temp_RxBuffer[2] = 16#00) AND NOT (Temp_RxBuffer[2] = 16#80) THEN
								STATE_nbReceptedChar:=(temp_RxBuffer[0] + (Temp_RxBuffer[1] * 256)) + 3;
								nErrId := ERROR_MESSAGE_CCB;	(*CCB incohérent*)
								nstepInError := 4;
								ErrDescription := 'FB_ClientDataExcha - Bad CCB';
								LOG_COM[0].ERR := ErrDescription;
								MEMCPY( ADR(LOG_COM[0].RX),ADR(Temp_RxBuffer),MAX_RXBUFFER_SIZE+1);	(*enregistrement dans le journal d'échange*)
								eStep := DATAEXCHA_STATE_ERROR;
							(*la longeur effective de la trame donnée par le premier octet  n'est pas cohérente avec la longueur attendue*)
							(*alors erreur*)
							ELSIF NOT ((temp_RxBuffer[0] + (Temp_RxBuffer[1] * 256) + 3) = NbExpectedChar) THEN
								STATE_nbReceptedChar:=(temp_RxBuffer[0] + (Temp_RxBuffer[1] * 256)) + 3;
								nErrId := ERROR_MESSAGE_LENGTH;	(*longueur trame incoérente*)
								nstepInError := 4;
								ErrDescription := 'FB_ClientDataExcha - Bad message length';
								LOG_COM[0].ERR := ErrDescription;
								MEMCPY( ADR(LOG_COM[0].RX),ADR(Temp_RxBuffer),MAX_RXBUFFER_SIZE+1);	(*enregistrement dans le journal d'échange*)
								eStep := DATAEXCHA_STATE_ERROR;
							ELSIF  (CbReceived >= nbExpectedChar) THEN	(*si le nombre de caractère reçu >= au nombre de caractère attendu*)
								(*Verification que la chaine recue comporte bien un caractère d'acquittement si le CCB = 0*)
								STATE_nbReceptedChar:=nbExpectedChar;
								IF NOT (Temp_RxBuffer[4] = 16#06) AND (Temp_RxBuffer[2] = 16#00) THEN
									STATE_nbReceptedChar:=(temp_RxBuffer[0] + (Temp_RxBuffer[1] * 256)) + 3;
									nErrId := ERROR_MISSING_ACK;	(*longueur trame incohérente*)
									nstepInError := 4;
									ErrDescription := 'FB_ClientDataExcha - Missing ACK';
									LOG_COM[0].ERR := ErrDescription;
									MEMCPY( ADR(LOG_COM[0].RX),ADR(Temp_RxBuffer),MAX_RXBUFFER_SIZE+1);	(*enregistrement dans le journal d'échange*)
									eStep := DATAEXCHA_STATE_ERROR;
								ELSE
									(*Calcul du CRC theorique*)
									Temp_Byte := 0;
										FOR I:=2 TO UDINT_TO_INT(nbExpectedChar-2) DO
											Temp_byte := Temp_Byte + Temp_RxBuffer[I];
										END_FOR
									(*si le CRC theorique n'est pas égal au CRC effectif alors erreur*)
									IF NOT (Temp_byte = temp_RxBuffer[NbExpectedChar-1])THEN
										STATE_nbReceptedChar:=(temp_RxBuffer[0] + (Temp_RxBuffer[1] * 256)) + 3;
										nErrId := ERROR_MESSAGE_LENGTH;	(*longueur trame incoérente*)
										nstepInError := 4;
										ErrDescription := 'FB_ClientDataExcha - Bad CRC';
										LOG_COM[0].ERR := ErrDescription;
										MEMCPY( ADR(LOG_COM[0].RX),ADR(Temp_RxBuffer),MAX_RXBUFFER_SIZE+1);	(*enregistrement dans le journal d'échange*)
										eStep := DATAEXCHA_STATE_ERROR;
										(*Tout est ok - on copy le buffer de réception temporaire dans le buffer de reception définitif*)
									ELSE
										MEMCPY(  ADR( RxBuffer ), ADR( Temp_rxBuffer ), NbExpectedChar); (*on récupère la chaine dans le buffer*)
										bBusy := FALSE;						(*Raz de l'indicateur de fonction d'émission/réception en cours*)
										VAR_COUNT_RETRY := 0; 				(*Raz du compteur de tentative de communication*)
										NErrId := 0;
										ErrDescription := 'NO ERROR ';
										nstepInError := 0;
										STATE_nbReceptedChar:=(temp_RxBuffer[0] + (Temp_RxBuffer[1] * 256)) + 3;
										eStep := DATAEXCHA_STATE_IDLE;
										LOG_COM[0].ERR := 'OK';
								 		MEMCPY( ADR(LOG_COM[0].RX),ADR(Temp_RxBuffer),NbExpectedChar);
									END_IF
								END_IF
							ELSE
								eStep := DATAEXCHA_STATE_RECEIVE_START; (* on répète l'étape de reception *)
							END_IF
						END_IF
					ELSE (* si il n'y a plus d'espace dispo dans le buffer *)
						nErrId := ERROR_RECEIVE_BUFFER_OVERFLOW;	(* buffer overflow !*)
						nstepInError := 4;
						ErrDescription := 'FB_ClientDataExcha - BUFFER OVERFLOW';
						LOG_COM[0].ERR := ErrDescription;
						MEMCPY( ADR(LOG_COM[0].RX),ADR(Temp_RxBuffer),MAX_RXBUFFER_SIZE+1);	(*enregistrement dans le journal d'échange*)
						eStep := DATAEXCHA_STATE_ERROR;
					END_IF

				ELSE(* sinon aucun bytes recus *)
					fbReceiveTON( PT := T#50ms); (* PRM_RECEIVE_POLLING_TIME );(* aucun  => on augmente la période de poolling *) *) (*TODO*)
					fbDisconnectTON( IN := TRUE, PT := PRM_RECEIVE_TIMEOUT );(* pas de reception => on active la tempo de timeout*)
					IF fbDisconnectTON.Q THEN (* si la tempo de timeout est écoulée*)
						fbDisconnectTON( IN := FALSE ); (*on désavtive la tempo de timeout*)
						(*LogError( 'FB_SocketReceive (local client)',  PLCPRJ_ERROR_RECEIVE_TIMEOUT );*)
						nStepInError := 4;
						ErrDescription := 'FB_ClientDataExcha - TIMEOUT ERROR';
						LOG_COM[0].ERR := ErrDescription;
						MEMCPY( ADR(LOG_COM[0].RX),ADR(Temp_RxBuffer),MAX_RXBUFFER_SIZE+1);	(*enregistrement dans le journal d'échange*)
						nErrID := ERROR_RECEIVE_TIMEOUT;
						eStep := DATAEXCHA_STATE_ERROR;
					ELSE(* si la tempo de timeout n'est pas écoulée *)
						eStep := DATAEXCHA_STATE_RECEIVE_START; (* on répète l'étape de reception *)
					END_IF
				END_IF
			ELSE(* si la fonction de reception renvoie une erreur*)
				nErrId := fbSocketReceive.nErrId;
				nStepInError := 4;
				ErrDescription := CONCAT('FB_ClientDataExcha - RECEIVE ERROR: ', UDINT_TO_STRING(nErrId));
				LOG_COM[0].ERR := ErrDescription;
				MEMCPY( ADR(LOG_COM[0].RX),ADR(Temp_RxBuffer),MAX_RXBUFFER_SIZE+1);	(*enregistrement dans le journal d'échange*)
				eStep := DATAEXCHA_STATE_ERROR;
			END_IF
		END_IF

	DATAEXCHA_STATE_ERROR:(* étape 5 - erreur *)
		VAR_COUNT_RETRY := VAR_COUNT_RETRY+1; (*incrémentation du compteur de tentative*)
		cbReceived := 0;	(*RAZ du nombre de donnée reçue*)
		IF VAR_COUNT_RETRY > 3 THEN	(*on accepte les 3 tentatives*)
			STATE_Com_Err_counter := STATE_Com_err_counter + 1;
			bError := TRUE;	(*mise à 1 du drapeau d'erreur*)
			bBusy := FALSE;	(*on reset le drapeau de fonction occupée*)
			eStep := DATAEXCHA_STATE_IDLE;	(*on retourne à l'étape 0*)
		ELSE (*sinon, on retente l'envoi aprés avoir purger le buffer de réception*)
			(*RAZ du buffer de réception et du buffer de réception temporaire*)
			FOR i:=0 TO UDINT_TO_INT(MAX_RXBUFFER_SIZE) DO
				Temp_RxBuffer[i] := 0;
				RxBuffer[i] :=0;
			END_FOR
			fbReceiveTON( IN := FALSE, PT := T#0s ); 	(* Réglage du buffer de réception à 0 pour lire asap *)
			fbDisconnectTON( IN := FALSE, PT := T#0s );	(* désactivation du timer de timeout *)
			eStep :=DATAEXCHA_STATE_RECEIVE_BEFORE_RETRY_START;
		END_IF


	DATAEXCHA_STATE_RECEIVE_BEFORE_RETRY_START:	(*etape 6 - vidage du buffer de recéption*)
		fbDisconnectTON(  );	(*lancement de la tempo de timeout : - désactivée sur cette étape*)
		fbReceiveTON( IN := TRUE,PT:=T#500ms );	(*temporisaton de 500 ms pour permettre à l'XTC de remplir le buffer de réception avant de relancer
												une requete*)
		IF fbReceiveTON.Q THEN
			fbReceiveTON( IN := FALSE );
			fbSocketReceive( bExecute := FALSE );
			fbSocketReceive(  hSocket:= hSocket,
						pDest:= ,	(*ajouté au buffer de réception à partir du dernier index CbReceived*)
						cbLen:= SIZEOF( Temp_rxBuffer ),   (*longueur max = longeur du buffer - dernier index CbReceived*)
						bExecute:= TRUE );
			eStep := DATAEXCHA_STATE_RECEIVE_BEFORE_RETRY_WAIT;
		END_IF
	DATAEXCHA_STATE_RECEIVE_BEFORE_RETRY_WAIT:	(*etape 7 - attente réponse*)
			fbSocketReceive( bExecute := FALSE );
			IF NOT fbSocketReceive.bBusy THEN		(*si pas fonction de réception en cours*)
				IF NOT  fbSocketReceive.bError THEN	(*si pas d'erreur*)
					fbReceiveTON( IN := FALSE, PT := T#0s ); 		(* Réglage du buffer de réception à 0 pour lire asap à la prochaine tentative *)
					fbDisconnectTON( IN := FALSE, PT := T#0s );		(* désactivation du timer de timeout *)
					eStep := DATAEXCHA_STATE_SEND_START;	(*on retente un envoi de requete*)
				ELSE(* si la fonction de reception renvoie une erreur*)
					nErrId := fbSocketReceive.nErrId;
					nStepInError := 7;
					eStep := DATAEXCHA_STATE_ERROR;			(*on retourne à la fonction de retentative*)
					ErrDescription := CONCAT('FB_ClientDataExcha - RECEIVE ERROR BEFORE RETRY: ', UDINT_TO_STRING(nErrId));
					SHIFT_BUFFER_DIALOG();
					LOG_COM[0].ERR := ErrDescription;

			END_IF
		END_IF
END_CASE

ACTION SHIFT_BUFFER_DIALOG:
(*Action de décalage du buffer de mémorisation des trames emises et recues dans le journal*)

(*on décale les lignes du buffer de com dans le journal des trames d'émission et réception*)
FOR I:= UDINT_TO_INT(MAX_BUFFER_DIALOG-1) TO 0 BY -1 DO
	LOG_COM[I+1].RX := LOG_COM[I].RX;
	LOG_COM[I+1].TX := LOG_COM[I].TX;
	LOG_COM[I+1].ERR := LOG_COM[I].ERR;
END_FOR
(*RAZ log en réception - ligne 0*)
FOR I:=0 TO UDINT_TO_INT(MAX_RXBUFFER_SIZE) BY 1 DO
	LOG_COM[0].RX[I] := 0;
END_FOR
(*RAZ log en émission - ligne 0*)
FOR I:=0 TO UDINT_TO_INT(MAX_TXBUFFER_SIZE) BY 1 DO
	LOG_COM[0].TX[I] := 0;
END_FOR
END_ACTION

END_FUNCTION_BLOCK

// ---- POUs/Fonction/FONCTION EFFLUVAGE/BLOCK_EFFLUVAGE.TcPOU
FUNCTION_BLOCK BLOCK_EFFLUVAGE
(* Fonction effluvage *)

(****************historique des versions*****************************)

(* Version 0-0 - SD - VERSION INITIALE EVA760 n°11 - 8152 *)
(* Version 1-0 - GV - Ajout arret automatique de sécurité si rotation en cours et pas porte*)

(*************************************************************************)

VAR_INPUT
(*information générale*)
	RESET:					BOOL;
	MANUAL:					BOOL;
	DOOR:					BOOL;	(*etat de fermeture des portes*)
	VAC:					BOOL;
	IN_Fin_Etape :			BOOL;
	CTRL_PLC:				BOOL;

(*Objet*)
	ALEFF:					ALIM_EFFLUVAGE;
(*Opérations *)
	OP_Marche_Eff:			BLOCK_OPERATION;
	OP_Arret_Eff:			BLOCK_OPERATION;
	OP_Gestion_Eff:			BLOCK_G7;

END_VAR
VAR_INPUT PERSISTENT
	PRM_TPS_effluvage:		TIME;			(*durée de l'effluvage*)
	PRM_consigne:			REAL;			(*Consigne de l'effluvage*)
	PRM_Tension_attendue:	REAL;			(*Tension attendue pour surveillance*)
	IsAssembly:				BOOL;			(*entité de type ensemble*)
	TagXml:					UINT;
	IdXml: 					STRING;
	IdParent: 				STRING;			(*MNEMO du pére*)
	MNEMO:					STRING;			(*MNEMO de cette entité *)
END_VAR

VAR_OUTPUT
	STATE_TEMPS_EFF:		TIME;				(*retour de temps d'effluvage*)
	STATE_TIMER_EC:			BOOL;				(*Tempo effluvage en cours*)
END_VAR

VAR
	TIMER_Effluvage:		TON;			(*Temporisation de l'effluvage*)
END_VAR

PRL();

(*appel des opérations*)
ACT_Arret_Eff();
ACT_Marche_Eff();

(*action en sortie*)
POST();

ACTION ACT_Arret_Eff:
(* OPERATION ARRET Effluvage*)
(* arrêt de l'effluvage*)

(*initialisation de l'opération*)
OP_Arret_Eff(
	CTRL_PLC:= CTRL_PLC,
	RESET:= RESET,
	ENABLE_INT:=TRUE,
	MANUAL:= MANUAL,
	ON_AUTO_INT:= ALEFF.DEF_Off_auto.DEF AND NOT MANUAL,
	RESTART_ENABLE_IF_OK:= FALSE,
	N_STEP_OP_OK:=3 ,
	N_STEP_OP_NOK:=0
	);


Op_arret_eff.PRL();

(*GRAFCET*)
(* initialisation du grafcet*)
IF 		OP_Arret_Eff.ETAPE = 0 THEN
				OP_Arret_Eff.ETAPE.0 := TRUE;
(*repositionnement sur étape 0*)
ELSIF	MANUAL OR
		OP_Marche_eff.Etape.1 OR
		RESET
					THEN

				OP_Arret_Eff.ETAPE := 0;			(*RAZ grafcet*)
				OP_Arret_Eff.ETAPE.0:=TRUE;
(*étape 0-1*)
ELSIF 	OP_Arret_Eff.ETAPE.0
			AND OP_Arret_Eff.MARCHE_OP
				THEN
				OP_Arret_Eff.ETAPE.1:=TRUE;
				OP_Arret_Eff.ETAPE.0:=FALSE;
(*étape 1-2*)
ELSIF	OP_Arret_Eff.ETAPE.1
		AND OP_Marche_Eff.etape.0 THEN
				OP_Arret_Eff.Etape.2:=TRUE;
				OP_Arret_Eff.Etape.1:=FALSE;
(*étape 2-3*)
ELSIF 	OP_Arret_Eff.Etape.2
			 THEN
				OP_Arret_Eff.Etape.3:=TRUE;
				OP_Arret_Eff.Etape.2:=FALSE;
END_IF;


(*cloture du traitement de l'opération*)
OP_Arret_Eff.POST();
END_ACTION

ACTION ACT_Gestion_Eff:
(*(* OPERATION gestion Effluvage*)
(*gestion global de l'effluvage de l'effluvage*)

(*initialisation de l'opération*)
OP_Gestion_Eff(
	N_STEP_OP_OK:=7,
	N_STEP_OP_NOK:=0 ,
	 );



(*GRAFCET*)
(* initialisation du grafcet*)
IF 		OP_Gestion_Eff.ETAPE = 0 THEN
				OP_Gestion_Eff.ETAPE.0 := TRUE;
(*repositionnement sur étape 0*)
ELSIF	MANUAL OR
		OP_Arret_eff.Etape.1 OR
		RESET
					THEN

				OP_Gestion_Eff.ETAPE := 0;			(*RAZ grafcet*)
				OP_Gestion_Eff.ETAPE.0:=TRUE;
(*étape 0-1*)
ELSIF 	OP_Gestion_Eff.ETAPE.0
			(*AND demande de marche d'effluvage*)
				OP_Gestion_Eff.ETAPE.1:=TRUE;
				OP_Gestion_Eff.ETAPE.0:=FALSE;
(*étape 1 ou 2 ou 3 ou 4 à 5*)
ELSIF IN_Recp_Fin_Etape
		 AND (OP_Gestion_Eff.ETAPE.1 OR OP_Gestion_Eff.ETAPE.2
				OR OP_Gestion_Eff.ETAPE.3 OR OP_Gestion_Eff.ETAPE.4)
		 THEN
				OP_Gestion_Eff.Etape.5:=TRUE;
				OP_Gestion_Eff.Etape.1:=FALSE;
				OP_Gestion_Eff.Etape.2:=FALSE;
				OP_Gestion_Eff.Etape.3:=FALSE;
				OP_Gestion_Eff.Etape.4:=FALSE;
(*étape 1-2*)
ELSIF	OP_Gestion_Eff.ETAPE.1
		AND PRG_POMPAGE.POMPAGE.OP_Marche_Pompes.OK AND TH_Pompage THEN
				OP_Gestion_Eff.Etape.2:=TRUE;
				OP_Gestion_Eff.Etape.1:=FALSE;

(*étape 2-3*)
ELSIF 	OP_Marche_Eff.Etape.2
		AND PRG_POMPAGE.POMPAGE.OP_Isolement.OK (*AND rotaion du Ps ok*)
			 THEN
				OP_Marche_Eff.Etape.3:=TRUE;
				OP_Marche_Eff.Etape.2:=FALSE;
(*étape 3-4*)
ELSIF 	OP_Gestion_Eff.Etape.3
		AND PRG_SERVITUDES.LIGNE_REF[2].STATE_Ok (*fonction gaz ligne de gaz 2 ok ??*)AND TH_Effluvage
			 THEN
				OP_Gestion_Eff.Etape.4:=TRUE;
				OP_Gestion_Eff.Etape.3:=FALSE;
(*étape 4-5*)
ELSIF 	OP_Gestion_Eff.Etape.4
		AND OP_Marche_Eff.OK
			 THEN
				OP_Gestion_Eff.Etape.5:=TRUE;
				OP_Gestion_Eff.Etape.4:=FALSE;
(*étape 5-6*)
ELSIF 	OP_Gestion_Eff.Etape.5
		AND OP_Arret_Eff.OK AND  PRG_SERVITUDES.LIGNE_REF[2].STATE_Ar (*fonction gaz ligne de gaz 2 à l'arret ??*)
			 THEN
				OP_Gestion_Eff.Etape.6:=TRUE;
				OP_Gestion_Eff.Etape.5:=FALSE;
(*étape 6-7*)
ELSIF 	OP_Gestion_Eff.Etape.6
		AND PRG_POMPAGE.POMPAGE.OP_Marche_Pompes.ok
			 THEN
				OP_Gestion_Eff.Etape.7:=TRUE;
				OP_Gestion_Eff.Etape.6:=FALSE;
END_IF;


(*cloture du traitement de l'opération*)
OP_Gestion_Eff.POST;*)
RETURN;
END_ACTION

ACTION ACT_Marche_Eff:
(* OPERATION Marche Effluvage*)


(*initialisation de l'opération*)
OP_Marche_Eff(
	CTRL_PLC:= CTRL_PLC,
	RESET:= RESET,
	ENABLE_INT:= DOOR AND VAC,
	MANUAL:= MANUAL,
	ON_AUTO_INT:= FALSE,
	RESTART_ENABLE_IF_OK:= FALSE,
	N_STEP_OP_OK:=4,
	N_STEP_OP_NOK:=0);

Op_marche_eff.PRL();

(*GRAFCET*)
(* initialisation du grafcet*)
IF 		OP_Marche_Eff.ETAPE = 0 THEN
				OP_Marche_Eff.ETAPE.0 := TRUE;
(*repositionnement sur étape 0*)
ELSIF	MANUAL OR
		OP_Arret_eff.Etape.1 OR
		RESET
					THEN

				OP_Marche_Eff.ETAPE := 0;			(*RAZ grafcet*)
				OP_Marche_Eff.ETAPE.0:=TRUE;
(*étape 0-1*)
ELSIF 	OP_Marche_Eff.ETAPE.0
			AND OP_Marche_Eff.MARCHE_OP
			THEN
				OP_Marche_Eff.ETAPE.1:=TRUE;
				OP_Marche_Eff.ETAPE.0:=FALSE;
(*étape 1-2*)
ELSIF	OP_Marche_Eff.ETAPE.1
		AND OP_Arret_Eff.etape.0 THEN
				OP_Marche_Eff.Etape.2:=TRUE;
				OP_Marche_Eff.Etape.1:=FALSE;
(*étape 2-3*)
ELSIF 	OP_Marche_Eff.Etape.2
		AND ALEFF.STATE_plasma
			 THEN
				OP_Marche_Eff.Etape.3:=TRUE;
				OP_Marche_Eff.Etape.2:=FALSE;
(*étape 3-4*)
ELSIF 	OP_Marche_Eff.Etape.3
		AND TIMER_Effluvage.q
			 THEN
				OP_Marche_Eff.Etape.4:=TRUE;
				OP_Marche_Eff.Etape.3:=FALSE;
(*étape 4-5*)
ELSIF 	OP_Marche_Eff.Etape.4
		AND ALEFF.STATE_OFF
			 THEN
				OP_Marche_Eff.Etape.0:=TRUE;
				OP_Marche_Eff.Etape.4:=FALSE;
END_IF;



(*cloture du traitement de l'opération*)
OP_Marche_Eff.POST();
END_ACTION

ACTION POST:
(********************************************************************************)
(*      MEFF :    Sortie TOR de pilotage du générateur d'effluvage        *)
(********************************************************************************)
IF OP_Marche_Eff.Etape.2
THEN
	ALEFF.CO_On		:= 	TRUE;
ELSIF OP_Marche_Eff.Etape.4 OR
		OP_Arret_Eff.Etape.2 OR
		OP_marche_eff.etape.0 AND OP_Arret_Eff.Etape.0
	THEN
	ALEFF.CO_ON	:= 	FALSE;
END_IF;


(*---------------------------------------------------------------------------------------------------------------------*)
(* consigne d'effluvage*)
IF  OP_Marche_Eff.Etape.2 OR OP_Marche_eff.Etape.3 OR
	 OP_marche_eff.Etape.4 OR MANUAL THEN
		ALEFF.PRM_Consigne := PRM_consigne;
		ALEFF.PRM_Tension_attendue := PRM_Tension_attendue;
ELSIF NOT MANUAL THEN
		ALEFF.PRM_Consigne := 0.0;
		ALEFF.PRM_Tension_attendue := 0.0;
END_IF


(***********************************************)
(*                Demande diverse                       *)
(***********************************************)
(*                Temporisations                            *)
(*            Tempo d'effluvage                          *)

TIMER_Effluvage	(
					PT:=PRM_TPS_Effluvage,
					IN:=OP_Marche_eff.Etape.3
					);
STATE_TEMPS_EFF := TIMER_Effluvage.ET;
STATE_TIMER_EC := OP_Marche_Eff.Etape.3;
ALeff(
	RESET:= RESET,
	MANUAL:=MANUAL ,
	DOOR:= DOOR,
	VAC:=VAC,
	EN_On_INT:=TRUE );
END_ACTION

ACTION PRL:
	OP_Marche_Eff.IdParent	:=	MNEMO;
	OP_Marche_Eff.MNEMO	:=	CONCAT(MNEMO,'_MARCHE');
	OP_Marche_Eff.IdXML		:=	'0';
	OP_Marche_Eff.TagXML	:=	1;

	OP_Arret_Eff.IdParent		:=	MNEMO;
	OP_Arret_Eff.MNEMO		:=	CONCAT(MNEMO,'_ARRET');
	OP_Arret_Eff.IdXML		:=	'0';
	OP_Arret_Eff.TagXML		:=	2;
END_ACTION

END_FUNCTION_BLOCK

// ---- POUs/Fonction/FONCTION PS/BLOCK_ROTATION_PS.TcPOU
FUNCTION_BLOCK BLOCK_ROTATION_PS
(* Fonction PS spécifique à l'affaire 8152 *)

(****************historique des versions*****************************)

(* Version 0-0 - SD - VERSION INITIALE EVA760 n°11 - 8152 *)
(* Version 1-0 - GV - Ajout arret automatique de sécurité si rotation en cours et pas porte*)

(*************************************************************************)

VAR_INPUT

(*information générale*)
	RESET:					BOOL;
	MANUAL:					BOOL;						 (*mode de fonctionnement de la fonction*)
	CTRL_PLC:				BOOL;
(* déclaration du moteur du PS*)
	MPS11:					BLOCK_VARIATEUR_MOTEUR;

(*sécurité*)
	DOOR:					BOOL;						(*information porte fermée*)
	INTERLOCK:				BOOL;						(*interlock de securité*)
(*opération*)
	OP_Rotation:			BLOCK_OPERATION;			(*opération rotation continue*)
	OP_Stop:				BLOCK_OPERATION;			(*opération arrêt*)
	(*Paramètre*)
	PRM_Vitesse:			REAL:=5;			 			(*Vitesse de rotation en mode rotation continue*)

END_VAR

VAR_INPUT PERSISTENT
(* Entité*)
	IsAssembly:				BOOL;						(*entité de type ensemble*)
	TagXml:					UINT;
	IdXml: 					STRING;
	IdParent: 				STRING;						(*MNEMO du pére*)
	MNEMO:					STRING;						(*MNEMO de cette entité *)

END_VAR

VAR_OUTPUT
	STATE_NOK:				BOOL;						(*Présence d'un défaut*)
END_VAR

VAR_IN_OUT
END_VAR

VAR
END_VAR

PRL();

ACT_ROTATION();
ACT_STOP();

POST();

ACTION ACT_ROTATION:
(* OPERATION rotation*)
(* Rotation continue du porte substrat*)

(*initialisation de l'opération*)
OP_Rotation(
	CTRL_PLC:= CTRL_PLC,
	RESET:= RESET,
	ENABLE_INT:= DOOR AND INTERLOCK ,
	MANUAL:= FALSE,
	ON_AUTO_INT:=FALSE,
	RESTART_ENABLE_IF_OK:= TRUE,
	N_STEP_OP_OK:=2,
	N_STEP_OP_NOK:=0);

(*appel de l'action de préparation de l'opération*)
OP_Rotation.PRL();


(*GRAFCET*)
(* initialisation du grafcet*)
IF 		OP_Rotation.Etape = 0
		THEN
				OP_Rotation.Etape.0 := TRUE;
(*repositionnement sur étape 0*)
ELSIF	RESET OR OP_Stop.ETAPE.1OR MANUAL
		THEN
				OP_Rotation.Etape := 0;			(*RAZ grafcet*)
				OP_Rotation.Etape.0  := TRUE;
(*étape 0-1*)
ELSIF 	OP_Rotation.Etape.0
		AND OP_Rotation.MARCHE_OP
		THEN
				OP_Rotation.Etape.1:=TRUE;
				OP_Rotation.Etape.0:=FALSE;
(*étape 1-2*)
ELSIF	OP_Rotation.Etape.1
		 AND OP_Stop.AR
		THEN
				OP_Rotation.Etape.2:=TRUE;
				OP_Rotation.Etape.1:=FALSE;
END_IF;
(*cloture du traitement de l'opération*)
OP_Rotation.POST();
END_ACTION

ACTION ACT_STOP:
(* OPERATION arrêt mouvement*)
(* Arrêt des mouvement de l'axe*)

(*initialisation de l'opération*)
OP_Stop(
	CTRL_PLC:= CTRL_PLC,
	RESET:= RESET,
	ENABLE_INT:= TRUE ,
	MANUAL:= FALSE,
	ON_AUTO_INT:= MPS11.DEF_Off_auto.DEF AND NOT MANUAL,
	RESTART_ENABLE_IF_OK:= TRUE,
	N_STEP_OP_OK:=2,
	N_STEP_OP_NOK:=0);

(*appel de l'action de préparation de l'opération*)
OP_Stop.PRL();


(*GRAFCET*)
(* initialisation du grafcet*)
IF 		OP_Stop.Etape = 0
		THEN
				OP_Stop.Etape.0 := TRUE;
(*repositionnement sur étape 0*)
	ELSIF	( OP_Rotation.Etape.1 OR RESET OR MANUAL )
		THEN
				OP_Stop.Etape := 0;			(*RAZ grafcet*)
				OP_Stop.Etape.0 := TRUE;
(*étape 0-1*)
	ELSIF 	OP_Stop.Etape.0
		AND OP_Stop.MARCHE_OP
		THEN
				OP_Stop.Etape.1:=TRUE;
				OP_Stop.Etape.0:=FALSE;
(*étape 1-2*)
	ELSIF	OP_Stop.Etape.1
		AND OP_Rotation.AR
		THEN
				OP_Stop.Etape.2:=TRUE;
				OP_Stop.Etape.1:=FALSE;
END_IF;
(*cloture du traitement de l'opération*)
OP_Stop.POST();
END_ACTION

ACTION POST:
(*************************************************************************)
(*      	    MPS11 :    Sortie TOR de pilotage du moteur du PS            *)
(*************************************************************************)
IF OP_Rotation.Etape.2 THEN
	MPS11.CO_On	:= 	TRUE;
ELSIF OP_Stop.Etape.2 OR
		(OP_STOP.Etape.0 AND OP_rotation.Etape.0) THEN
	MPS11.CO_On	:= 	FALSE;
END_IF;

IF OP_rotation.Etape.2 OR OP_rotation.Etape.3 THEN
	MPS11.PRM_Cons_Vitesse := PRM_Vitesse;
END_IF


MPS11(
	RESET:= RESET,
	MANUAL:= MANUAL,
	DOOR:=DOOR ,
	EN_On_INT:=TRUE ,
	EN_Off_INT:= TRUE,
	CONF_EN_On:= 1,
	CONF_No_Safety_Auto:=FALSE  );


(*Codage des états*)
STATE_Nok		:=  OP_STOP.DEF_AUTO_ON.DEF OR OP_STOP.DEF_ON_REJECTED.DEF OR
					OP_ROTATION.DEF_AUTO_ON.DEF OR OP_ROTATION.DEF_ON_REJECTED.DEF OR MPS11.STATE_Nok;
END_ACTION

ACTION PRL:
(*commentaire pour les opérations*)
(* Mnémonique*)
MPS11.MNEMO := 'MPS11';
MPS11.IdParent := MNEMO;


(*commentaire dans les dictionnaires*)
IdXml 						:='5';
TagXml						:=0;

OP_Rotation.IdXml			:='6';
OP_Rotation.TagXml			:=2;

OP_Stop.IdXml				:='0';
OP_Stop.TagXml				:=2;
END_ACTION

END_FUNCTION_BLOCK

// ---- POUs/Fonction/FONCTIONS GAZ/BLOCK_LIGNE_GAZ_2_VANNES.TcPOU
FUNCTION_BLOCK BLOCK_LIGNE_GAZ_2_VANNES
(* Gestion d'une ligne de gaz avec deux vannes et un debitmètre *)

VAR_INPUT
(*informations générales*)
	RESET:					BOOL;		(* Condition de réinitialisation de la fonction *)
	MANUAL:					BOOL;		(* Ordre de commmande manuel de la fonction *)
	CTRL_PLC:				BOOL;		(* Mode de contrôle de la fonction - 0 = contrôle depuis l'IHM - 1=contrôle depuis l'automate*)
(*sécurité*)
	VAC:					BOOL;		(* Entrée d'interlock de vide*)
	DOOR:					BOOL;		(* Entrée d'interlock porte*)
(*Composants*)
	VGI1:					BLOCK_ACTUATOR2;				(* Vanne injection de gaz de la ligne*)
	VGI2:					BLOCK_ACTUATOR2	;				(*Seconde vanne d'injection de la ligne*)

(*Paramètres*)
	PRM_Disable_Surv:		BOOL;		(* Désactivation surveillance débit externe au bloc *)
	PRM_Flow:				REAL;		(* ~ (OPC : 1 : available for OPC-clients) *)	(* Consigne de débit gaz*)
	CO_Modif:				BOOL;		(* Demande modification en ligne*)
(*Opérations*)
	OP_MARCHE:				BLOCK_OPERATION;		(* Opération mise en gaz ligne*)
	OP_ARRET:				BLOCK_OPERATION;		(* Opération arret gaz*)
	OP_RAMPE:				BLOCK_RAMP;				(* Opération rampe de gaz*)
END_VAR

VAR_OUTPUT
	STATE_NOK:				BOOL;		(* Défaut ligne de gaz*)
	STATE_Ready:			BOOL;		(* Mise en gaz autorisée*)
	O_SURV_DISABLE:			BOOL;		(* I_STANDARD -- Sortie de désactivation de la surveillance du débit vers le bloc MFC associé*)
END_VAR

VAR_INPUT PERSISTENT
	(*Entité*)
	IsAssembly:		BOOL;			(*entité : fonction*)
	IdXML:			STRING;			(*nom entité : identifiant pour recherche dans dico*)
	TagXML:			UINT;			(*nom entité : identifiant pour recherche dans dico*)
	IdParent:		STRING;			(*MNEMO de l'appelant*)
	MNEMO:			STRING;			(*MNEMO de l'entité*)
END_VAR

VAR_IN_OUT
	DG_PRM_FLOW:			REAL;											(*Variable PRM flow du massflow associé*)
END_VAR

VAR
	FM_CO_Modif:			R_TRIG;
	VAR_Flow:				REAL;
END_VAR

(*Début de bloc*)
PRL();
(*Opération arrêt gaz*)
ACT_STOP();
(*Opération marche gaz*)
ACT_START();
(*Fin de bloc*)
POST();

ACTION ACT_START:
(*OPERATION MARCHE GAZ*)
(*Marche gaz en continu*)

OP_MARCHE(
	CTRL_PLC:= CTRL_PLC,
	RESET:= reset,
	MANUAL:=manual ,
	RESTART_ENABLE_IF_OK:=TRUE ,
	N_STEP_OP_OK:= 3,
	N_STEP_OP_NOK:=0 );

(*appel de l'action de préparation de l'opération*)
OP_MARCHE.PRL();

(*GRAFCET*)
(* initialisation du grafcet*)
IF 		OP_MARCHE.ETAPE = 0
		THEN
				OP_MARCHE.ETAPE.0 := TRUE;
(*repositionnement sur étape 0*)
ELSIF 	MANUAL OR RESET OR OP_ARRET.ETAPE.1
		THEN
				OP_MARCHE.ETAPE := 0;
				OP_MARCHE.ETAPE.0:=TRUE;
(*étape 0-1*)
ELSIF 	OP_MARCHE.ETAPE.0 AND OP_MARCHE.MARCHE_OP
		THEN
				OP_MARCHE.ETAPE.1:=TRUE;
				OP_MARCHE.ETAPE.0:=FALSE;
(*étape 1-2*)
ELSIF	OP_MARCHE.ETAPE.1 AND OP_ARRET.ETAPE.0
		THEN
				OP_MARCHE.ETAPE.2:=TRUE;
				OP_MARCHE.ETAPE.1:=FALSE;
(*étape 2-3*)
ELSIF	OP_MARCHE.ETAPE.2 AND ((VGI1.STATE_On AND VGI2.STATE_On) OR VAR_Flow=0)
		THEN
				OP_MARCHE.ETAPE.3:=TRUE;
				OP_MARCHE.ETAPE.2:=FALSE;
(*étape 3-2*)
ELSIF	OP_MARCHE.ETAPE.3 AND
	(OP_MARCHE.MARCHE_OP OR  (FM_CO_Modif.Q AND NOT OP_RAMPE.MARCHE.EC))
		THEN
				OP_MARCHE.ETAPE.2:=TRUE;
				OP_MARCHE.ETAPE.3:=FALSE;
END_IF;
(*cloture du traitement de l'opération*)
OP_MARCHE.POST();
END_ACTION

ACTION ACT_STOP:
(*OPERATION STOP GAZ*)

OP_ARRET(
	CTRL_PLC:= CTRL_PLC,
	RESET:= reset,
	MANUAL:=manual ,
	RESTART_ENABLE_IF_OK:=FALSE ,
	N_STEP_OP_OK:= 2,
	N_STEP_OP_NOK:=0 );

(*appel de l'action de préparation de l'opération*)
OP_ARRET.PRL();

(*GRAFCET*)
(* initialisation du grafcet*)
IF 		OP_ARRET.ETAPE = 0
		THEN
				OP_ARRET.ETAPE.0 := TRUE;
(*repositionnement sur étape 0*)
ELSIF 	MANUAL OR RESET OR OP_MARCHE.ETAPE.1
		THEN
				OP_ARRET.ETAPE := 0;
				OP_ARRET.ETAPE.0:=TRUE;
(*étape 0-1*)
ELSIF 	OP_ARRET.ETAPE.0 AND OP_ARRET.MARCHE_OP
		THEN
				OP_ARRET.ETAPE.1:=TRUE;
				OP_ARRET.ETAPE.0:=FALSE;
(*étape 1-2*)
ELSIF 	OP_ARRET.ETAPE.1 AND VGI1.STATE_OFF AND VGI2.STATE_Off AND OP_MARCHE.Etape.0
		THEN
				OP_ARRET.ETAPE.2:=TRUE;
				OP_ARRET.ETAPE.1:=FALSE;
END_IF;

(*cloture du traitement de l'opération*)
OP_ARRET.POST();
END_ACTION

ACTION POST:
(*Etat prêt*)
STATE_READY	:=	(*VAC AND*) DOOR;

(*Autorisations*)
OP_ARRET.ON_AUTO_INT	:=	VGI1.DEF_Off_auto.DEF OR VGI2.DEF_Off_auto.DEF AND NOT Manual;
OP_ARRET.ENABLE_INT		:=	TRUE;
OP_MARCHE.ENABLE_INT	:=	STATE_Ready;

(*Gestion demandes*)
FM_CO_Modif(clk:=CO_modif);

(*Gestion rampe*)
IF	FM_CO_Modif.Q AND OP_RAMPE.MARCHE.EC THEN
	OP_RAMPE.CO_Modif_Rampe	:=	TRUE;
END_IF;
OP_RAMPE.MARCHE.RESET		:=	NOT OP_MARCHE.OK;
OP_RAMPE.MARCHE.ENABLE_INT	:=	OP_MARCHE.OK;
OP_RAMPE.MARCHE.CTRL_PLC 	:= CTRL_PLC;
OP_RAMPE(
	IN_VALUE:=DG_PRM_FLOW,
	PRM_RAMPE:=PRM_Flow);

(*Gestion vanne n°1*)
VGI1.CO_On	:= 	(OP_MARCHE.Etape.2 OR OP_MARCHE.Etape.3) AND (DG_PRM_FLOW>0);
VGI1(
	RESET:=Reset ,
	MANUAL:=Manual ,
	EN_On_INT:=STATE_Ready);

(*Gestion vanne n°2*)
VGI2.CO_On	:= 	(OP_MARCHE.Etape.2 OR OP_MARCHE.Etape.3) AND (DG_PRM_FLOW>0);
VGI2(
	RESET:=Reset ,
	MANUAL:=Manual ,
	EN_On_INT:=STATE_Ready);


(*Gestion débitmètre*)
IF		OP_MARCHE.Etape.2 THEN
	DG_PRM_FLOW	:=	PRM_Flow;
ELSIF	OP_MARCHE.AR AND NOT manual THEN
	DG_PRM_FLOW	:=	0.0;
ELSIF	Manual THEN
	DG_PRM_FLOW	:=	PRM_Flow;
ELSIF	OP_RAMPE.MARCHE.EC THEN
	DG_PRM_FLOW	:=	OP_RAMPE.OUT_VALUE;
END_IF

(*Gestion défauts*)
(*alarme, défaut surveillance*)
O_SURV_DISABLE		:=	(NOT VGI1.STATE_On AND NOT VGI2.STATE_On) OR PRM_Disable_Surv;

(*Etat défaut*)
STATE_NOK		:=	FALSE;

(*Reset demandes*)
CO_Modif	:=	FALSE;
END_ACTION

ACTION PRL:
	OP_MARCHE.IdParent	:=	MNEMO;
	OP_MARCHE.MNEMO		:=	CONCAT(MNEMO,'_MARCHE');
	OP_MARCHE.IdXML		:=	'0';
	OP_MARCHE.TagXML	:=	1;

	OP_ARRET.IdParent	:=	MNEMO;
	OP_ARRET.MNEMO		:=	CONCAT(MNEMO,'_ARRET');
	OP_ARRET.IdXML		:=	'0';
	OP_ARRET.TagXML		:=	2;

	OP_RAMPE.IdParent	:=	MNEMO;
	OP_RAMPE.MNEMO		:=	CONCAT(MNEMO,'_RAMPE');
	OP_RAMPE.IdXML		:=	'18';
	OP_RAMPE.TagXML		:=	1;

	VGI1.IdXML					:=	'1';
	VGI1.TagXML					:=	1;
	VGI1.IdParent				:=	MNEMO;
	VGI1.DEF_Off_auto.IdXML		:=	'3';
	VGI1.DEF_Off_auto.TagXML	:=	11;
	VGI1.DEF_Off_Imposs.IdXML	:=	'3';
	VGI1.DEF_Off_Imposs.TagXML	:=	9;
	VGI1.DEF_On_Imposs.IdXML	:=	'3';
	VGI1.DEF_On_Imposs.TagXML	:=	6;

	(*TOCHECK*)
	VGI2.IdXML					:=	'1';
	VGI2.TagXML					:=	1;
	VGI2.IdParent				:=	MNEMO;
	VGI2.DEF_Off_auto.IdXML		:=	'3';
	VGI2.DEF_Off_auto.TagXML	:=	11;
	VGI2.DEF_Off_Imposs.IdXML	:=	'3';
	VGI2.DEF_Off_Imposs.TagXML	:=	9;
	VGI2.DEF_On_Imposs.IdXML	:=	'3';
	VGI2.DEF_On_Imposs.TagXML	:=	6;
END_ACTION

END_FUNCTION_BLOCK

// ---- POUs/Fonction/FONCTIONS GAZ/BLOCK_LIGNE_GAZ_NO_DG.TcPOU
	FUNCTION_BLOCK BLOCK_LIGNE_GAZ_NO_DG
(* Gestion d'une ligne de gaz avec une vanne et pas de débimètre *)

(****************historique des versions*****************************)

(* Version 1-0 - GV - VERSION INITIALE - Gestion d'une ligne de gaz sans débimètre - 8650*)
(* Version 2-0 - GV - Adaptation pour journal des évènements externe - 9070 - 07/2015*)

(*************************************************************************)

VAR_INPUT
(*informations générales*)
	RESET:					BOOL;		(* Condition de réinitialisation de la fonction *)
	MANUAL:				BOOL;		(* Ordre de commmande manuel de la fonction *)
	CTRL_PLC:				BOOL;		(* Mode de contrôle de la fonction - 0 = contrôle depuis l'IHM - 1=contrôle depuis l'automate*)
(*sécurité*)
	VAC:					BOOL;		(* Entrée d'interlock de vide*)
	DOOR:					BOOL;		(* Entrée d'interlock porte*)
(*Composants*)
	VGI:						BLOCK_ACTUATOR2;				(* Vanne injection de gaz de la ligne*)

(*Opérations*)
	OP_MARCHE:			BLOCK_OPERATION;		(* Opération mise en gaz ligne*)
	OP_ARRET:				BLOCK_OPERATION;		(* Opération arret gaz*)
END_VAR

VAR_OUTPUT
	STATE_NOK:				BOOL;		(* ~ (OPC : 1 : available for OPC-clients) *)	(* Défaut ligne de gaz*)
	STATE_Ready:			BOOL;		(* ~ (OPC : 1 : available for OPC-clients) *)	(* Mise en gaz autorisée*)
END_VAR

VAR_INPUT PERSISTENT
	(*Entité*)
	IsAssembly:		BOOL;			(*entité : fonction*)
	IdXML:			STRING;			(*nom entité : identifiant pour recherche dans dico*)
	TagXML:			UINT;			(*nom entité : identifiant pour recherche dans dico*)
	IdParent:			STRING;			(*MNEMO de l'appelant*)
	MNEMO:			STRING;			(*MNEMO de l'entité*)
END_VAR

(*Début de bloc*)
PRL();
(*Opération arrêt gaz*)
ACT_STOP();
(*Opération marche gaz*)
ACT_START();
(*Fin de bloc*)
POST();

ACTION ACT_START:
(*OPERATION MARCHE GAZ*)
(*Marche gaz en continu*)

OP_MARCHE(
	CTRL_PLC:= CTRL_PLC,
	RESET:= reset,
	MANUAL:=manual ,
	RESTART_ENABLE_IF_OK:=TRUE ,
	N_STEP_OP_OK:= 3,
	N_STEP_OP_NOK:=0 );

(*appel de l'action de préparation de l'opération*)
OP_MARCHE.PRL();

(*GRAFCET*)
(* initialisation du grafcet*)
IF 		OP_MARCHE.ETAPE = 0
		THEN
				OP_MARCHE.ETAPE.0 := TRUE;
(*repositionnement sur étape 0*)
ELSIF 	MANUAL OR RESET OR OP_ARRET.ETAPE.1
		THEN
				OP_MARCHE.ETAPE := 0;
				OP_MARCHE.ETAPE.0:=TRUE;
(*étape 0-1*)
ELSIF 	OP_MARCHE.ETAPE.0 AND OP_MARCHE.MARCHE_OP
		THEN
				OP_MARCHE.ETAPE.1:=TRUE;
				OP_MARCHE.ETAPE.0:=FALSE;
(*étape 1-2*)
ELSIF	OP_MARCHE.ETAPE.1 AND OP_ARRET.ETAPE.0
		THEN
				OP_MARCHE.ETAPE.2:=TRUE;
				OP_MARCHE.ETAPE.1:=FALSE;
(*étape 2-3*)
ELSIF	OP_MARCHE.ETAPE.2 AND VGI.STATE_On
		THEN
				OP_MARCHE.ETAPE.3:=TRUE;
				OP_MARCHE.ETAPE.2:=FALSE;
(*étape 3-2*)
ELSIF	OP_MARCHE.ETAPE.3 AND OP_MARCHE.MARCHE_OP
		THEN
				OP_MARCHE.ETAPE.2:=TRUE;
				OP_MARCHE.ETAPE.3:=FALSE;
END_IF;
(*cloture du traitement de l'opération*)
OP_MARCHE.POST();
END_ACTION

ACTION ACT_STOP:
(*OPERATION STOP GAZ*)

OP_ARRET(
	CTRL_PLC:= CTRL_PLC,
	RESET:= reset,
	MANUAL:=manual ,
	RESTART_ENABLE_IF_OK:=FALSE ,
	N_STEP_OP_OK:= 2,
	N_STEP_OP_NOK:=0 );

(*appel de l'action de préparation de l'opération*)
OP_ARRET.PRL();

(*GRAFCET*)
(* initialisation du grafcet*)
IF 		OP_ARRET.ETAPE = 0
		THEN
				OP_ARRET.ETAPE.0 := TRUE;
(*repositionnement sur étape 0*)
ELSIF 	MANUAL OR RESET OR OP_MARCHE.ETAPE.1
		THEN
				OP_ARRET.ETAPE := 0;
				OP_ARRET.ETAPE.0:=TRUE;
(*étape 0-1*)
ELSIF 	OP_ARRET.ETAPE.0 AND OP_ARRET.MARCHE_OP
		THEN
				OP_ARRET.ETAPE.1:=TRUE;
				OP_ARRET.ETAPE.0:=FALSE;
(*étape 1-2*)
ELSIF 	OP_ARRET.ETAPE.1 AND VGI.STATE_OFF AND OP_MARCHE.Etape.0
		THEN
				OP_ARRET.ETAPE.2:=TRUE;
				OP_ARRET.ETAPE.1:=FALSE;
END_IF;

(*cloture du traitement de l'opération*)
OP_ARRET.POST();
END_ACTION

ACTION POST:
(*Etat prêt*)
STATE_READY	:=	VAC AND DOOR;

(*Autorisations*)
OP_ARRET.ON_AUTO_INT	:=	VGI.DEF_Off_auto.DEF AND NOT Manual;
OP_ARRET.ENABLE_INT		:=	TRUE;
OP_MARCHE.ENABLE_INT	:=	STATE_Ready;

(*Gestion vanne*)
VGI.CO_On	:= 	(OP_MARCHE.Etape.2 OR OP_MARCHE.Etape.3);
VGI(
	RESET:=Reset ,
	MANUAL:=Manual ,
	EN_On_INT:=STATE_Ready);

(*Etat défaut*)
STATE_NOK		:=	FALSE;
END_ACTION

ACTION PRL:
	OP_MARCHE.IdParent		:=	MNEMO;
	OP_MARCHE.MNEMO			:=	CONCAT(MNEMO,'_MARCHE');
	OP_MARCHE.IdXML			:=	'0';
	OP_MARCHE.TagXML		:=	1;

	OP_ARRET.IdParent		:=	MNEMO;
	OP_ARRET.MNEMO			:=	CONCAT(MNEMO,'_ARRET');
	OP_ARRET.IdXML			:=	'0';
	OP_ARRET.TagXML			:=	2;

	VGI.IdXML					:=	'1';
	VGI.TagXML					:=	1;
	VGI.IdParent					:=	MNEMO;
	VGI.DEF_Off_auto.IdXML		:=	'3';
	VGI.DEF_Off_auto.TagXML		:=	11;
	VGI.DEF_Off_Imposs.IdXML		:=	'3';
	VGI.DEF_Off_Imposs.TagXML	:=	9;
	VGI.DEF_On_Imposs.IdXML		:=	'3';
	VGI.DEF_On_Imposs.TagXML	:=	6;
END_ACTION

END_FUNCTION_BLOCK

// ---- POUs/Fonction/FONCTIONS POMPAGE/BLOCK_POMP_1E_PCR_PPM_ASS_ETHERCAT.TcPOU
FUNCTION_BLOCK BLOCK_POMP_1E_PCR_PPM_ASS_ETHERCAT

(* Historique des versions*)
(* VERSION 1.0 - 05/2015 - GV - affaire 9070*)
(* VERSION 2.0 - 10/2022 - GV - ajout gestion roots *)


(* BLOCK GESTION POMPAGE CRYO ON BOARD ENCEINTE *)
(*	Gestion pompage enceinte sans sas constitué de :
	Pompe primaire pour prévidage, regen cryo et pompage interjoint
	Pompe cryogénique on-board CTI pour le pompage secondaire
	Vanne de pompage primaire enceinte
	Vanne de remise à atmosphère enceinte
	Vanne de pompage inter-joint (optionnelle)
	Vanne secondaire asservie, pilotée par ethercatf
*)

VAR_INPUT
(*information générale*)
	RESET:					BOOL;
	MANUAL:					BOOL;
	CTRL_PLC:				BOOL;
	I_Prep_Ventil_Ok:		BOOL;		(*information externe indiquant que l'enceinte est prête à être ventilée par ex. circulation d'eau à l'arrêt
										ou polycold arreté ou basculement en eau chaude ok ...*)
	I_Fin_Ventil:			BOOL;		(*information externe de fin de ventilation de l'enceinte  *)
	I_Stop_Mesure_OK:		BOOL;		(*information externe indiquant que les jauges ont été stoppées prélablement à la ventilation de l'enceinte*)
	IN_Pressure_RP:			REAL;		(*interfaçage avec M11.state_pression du PRG correspondant*)
	I_Ref_OK:				BOOL;		(*information externe indiquant que le refroidissement est ok pour démarrer les pompes*)
	
(*Gestion régen partielle*)
	IN_Temp_Etage1:			REAL;
	PRM_Temp_Post_Purge:	REAL;
	PRM_Tim_Post_Purge:		TIME;

(*Paramètres et commandes du test de remontée de pression*)
	PRM_Pr_test:			REAL;		(*Pression initiale de test de remontée*)
	PRM_Tim_test:			TIME;		(*Durée d'attente en test*)
	CO_Stop_Test_RP:		BOOL;		(*Demande arrêt test remontée de pression*)

(*sécurité*)
	IN_FE11T:				BOOL;		(*indicateur enceinte fermée - capteur 1*)
	IN_FE12T:				BOOL;		(*indicateur enceinte fermée - capteur 2*)
	IN_VT11F:				BOOL;		(*clapet SAS enceinte fermé*)

(*seuil de vide*)
	TH_Vide_Primaire:		BOOL;		(*Pression enceinte <= Seuil de fin de pompage primaire*)
	TH_Grosse_Fuite:		BOOL;		(*Pression enceinte <= Seuil de detection de grosse fuite enceinte*)
	TH_Atm:					BOOL;		(*pression enceinte >= Seuil pression atm. de fin de ventilation*)
	TH_RP_Enc:				BOOL;		(*pression enceinte <= Pression max. dans l'enceinte*)
	TH_Test_RP:				BOOL;		(*Pression <= Seuil de pression de test*)

(*composant de la fonction*)
	VP11:					BLOCK_ACTUATOR;									(*vanne de pompage primaire enceinte *)
	VH11:					BLOCK_ACTUATOR;									(*vanne de ventilation de l'enceinte*)
	PP11:					BLOCK_PPM;										(*Pompe primaire enceinte*)
	PR11:					BLOCK_PPM;										(*Pompe roots enceinte*)
	PS11:					BLOCK_PCR_CTI_OB;								(*Pompe cryogénique on board  enceinte*)
	VS11:					BLOCK_VVAT_653_ETHERCAT;						(*Vanne secondaire asservie pompage enceinte*)
	VINT:					BLOCK_ACTUATOR;									(*Vanne de pompage dans les interjoints*)

(*défaut*)
	DEF_PPrim:				PRCDEF;										(*défaut temps de pompage primaire dans l'enceinte*)
	DEF_Vent:				PRCDEF;										(*défaut temps de ventilation enceinte*)
	DEF_RP_enc:				PRCDEF;	 									(*défaut perte seuil de pompage primaire en pompage secondaire*)
	DEF_TGF:				PRCDEF;										(*défaut détection trés grosse fuite*)

(*opération*)
	OP_Marche_Pompes:			BLOCK_OPERATION;								(*opération marche pompe*)
	OP_Arret_Pompes:			BLOCK_OPERATION;								(*opération arrêt pompe*)
	OP_Isolement:				BLOCK_OPERATION;								(*opération stand-by*)
	OP_Ventilation:				BLOCK_OPERATION;								(*opération ventilation*)
	OP_Pompage_Sec:				BLOCK_OPERATION;								(*opération pompage secondaire*)
	OP_Pompage_Prim:			BLOCK_OPERATION;								(*opération pompage primaire*)
	OP_Pompage_Proc:			BLOCK_OPERATION;								(*opération pompage en procédé*)
	OP_Purge:					BLOCK_OPERATION;								(*opération purge*)
	OP_Regen:					BLOCK_OPERATION;								(*opération régénération pompe cryogénique*)
	OP_Regen_Part:				BLOCK_OPERATION;								(*opération de régénération partielle pompe cryogénique*)
	OP_Test_RP:					BLOCK_OPERATION;								(*opération test RP*)
	G7_pompage_interjoint:		BLOCK_G7;

END_VAR

VAR_INPUT PERSISTENT
(*paramètre*)
	PRM_Tim_SurVentil_E:		TIME;	(*durée du temps de surventilation*)
	PRM_Tim_Purge:				TIME;	(*durée du maintien pompage primaire en purge*)
	PRM_Tim_Arret_PP11:			TIME;	(*durée avant arrêt de la pompe primaire*)
	PRM_Pr_Atm:					REAL;	(*Pression atmosphérique dans l'enceinte*)
	PRM_Pr_PPrim:				REAL;	(*Pression de fin de pompage primaire dans l'enceinte*)
	PRM_Pr_RP_PPrim:			REAL;	(*Pression max admissible dans l'enceinte en pompage secondaire dans l'enceinte*)
	PRM_Pr_TGF:					REAL;	(*Pression de détection trés grosse fuite dans l'enceinte*)
	PRM_N_Purge:				USINT;	(*Nombre de cycles de purge pompage/ventilation*)
	CONF_Pompage_interjoint:	BOOL;	(*Utilisation de la pompe primaire pour le pompage interjoint sur l'enceinte*)
	CONF_VINT:					BOOL;	(*Utilisation d'une vanne d'isolement sur le pompage interjoint*)
	CONF_Volume_Enceinte:		REAL;	(*Volume pour RP*)

	PRM_Tim_Prep_Ventil:		TIME;	(*temporisation de prép ventilation (eau chaude suffisemment longtemps) *)

	(*Entité*)
	IsAssembly:		BOOL;		(*entité : ensemble*)
	IdXML:			STRING;		(*nom entité : identifiant pour recherche dans dico*)
	TagXML:			UINT;		(*nom entité : identifiant pour recherche dans dico*)
	IdParent:		STRING;		(*MNEMO de l'appelant*)
	MNEMO:			STRING;		(*MNEMO de l'entité*)
END_VAR


VAR_OUTPUT
	RQ_Prep_Ventil_Enc:		BOOL;											(*demande de préparation avant ventilation (réchauffement, arrêt eau ....*)
	RQ_Stop_Mesure_Enc:		BOOL;											(*demande d'arrêt de la mesure avant ventilation - Les blocs jauges concernés utilise
																			cette information pour stoppée les jauges préalablement à la ventilation*)
END_VAR

VAR_IN_OUT
END_VAR

VAR
	VAR_Reset_Sortie:					BOOL;
	TIMER_SurVentilation_Enc:			TON;		(*Temporistion de surventilation enceinte*)
	TIMER_Purge:						TON;		(*Temporisation de maintien pompage primaire en purge*)
	TIMER_Pompage_Interjoint:			TON;		(*Temporisation d'ouverture de la vanne de pompage interjoint*)
	TIMER_Arret_Roots:					TON;		(*Temporisation arrêt roots après prévidage*)
	TIMER_Arret_PP11:					TON;		(*Temporisation arrêt pompe primaire*)
	VAR_mem_isolement:					BOOL;
	VAR_Iter_Purge:						USINT;

	(*Pour RP*)
	VAR_Mem_Pression_Deb:		REAL;
	VAR_Mem_Pression_Fin:		REAL;
	VAR_Indicateur_Test:		REAL; 		(*résultat final*)
	TIMER_attente_test:			TON;		(*Temporisation pour test de remontée en pression*)
	FM_etape4:					R_TRIG;

	(*Pour prep ventil*)
	TIM_Prep_ventil:			TON;		(*timer de préparation ventil*)

	(*Pour regen*)
	FM_REGEN:						R_TRIG;		(* FM pompe cryogénique en régénération*)
	FD_REGEN:						F_TRIG;		(* FD pompe cryogénique en régénération*)
	TIMER_Post_Purge:				TON;		(*tempo max attente de retombée température après purge en regen partielle*)
	TIMER_etape6_regen:				TON;
END_VAR

PRL();

(*appel des opérations*)
ACT_ARRET_POMPES();
ACT_ISOLEMENT();
ACT_MARCHE_POMPES();
ACT_POMPAGE_PRIM();
ACT_POMPAGE_PROC();
ACT_POMPAGE_SEC();
ACT_VENTILATION();
ACT_PURGE();
ACT_REGEN();
ACT_REGEN_PART();
ACT_TEST_RP();
ACT_POMPAGE_INTERJOINT();

(*action en sortie*)
POST();

ACTION ACT_ARRET_POMPES:
(* OPERATION ARRET POMPES*)
(* arrêt des pompes*)

(*initialisation de l'opération*)
OP_ARRET_POMPES(
	CTRL_PLC:= CTRL_PLC,
	RESET:= RESET,
	ENABLE_INT:=TRUE,
	MANUAL:= MANUAL,
	ON_AUTO_INT:= (PP11.STATE_NOK AND PR11.STATE_NOK) AND (NOT OP_Pompage_Prim.Etape.0 OR NOT OP_Purge.Etape.0),
	RESTART_ENABLE_IF_OK:= FALSE,
	N_STEP_OP_OK:= 5,
	N_STEP_OP_NOK:=0);

(*appel de l'action de préparation de l'opération*)
OP_ARRET_POMPES.PRL();


(*GRAFCET*)
(* initialisation du grafcet*)
IF 		OP_Arret_Pompes.ETAPE = 0 THEN
				OP_Arret_Pompes.ETAPE.0 := TRUE;
(*repositionnement sur étape 0*)
ELSIF	MANUAL OR RESET OR OP_Marche_Pompes.ETAPE.1 THEN
				OP_Arret_Pompes.ETAPE := 0;			(*RAZ grafcet*)
				OP_Arret_Pompes.ETAPE.0:=TRUE;
(*étape 0-1*)
ELSIF 	OP_Arret_Pompes.ETAPE.0
		AND OP_Arret_Pompes.MARCHE_OP THEN
				OP_Arret_Pompes.ETAPE.1:=TRUE;
				OP_Arret_Pompes.ETAPE.0:=FALSE;
(*étape 1-2*)
ELSIF	OP_Arret_Pompes.ETAPE.1
		AND OP_Marche_Pompes.ETAPE.0  THEN
				OP_Arret_Pompes.Etape.2:=TRUE;
				OP_Arret_Pompes.Etape.1:=FALSE;
(*étape 2-3*)
ELSIF 	OP_Arret_Pompes.Etape.2
		AND (OP_Isolement.OK OR VAR_mem_isolement)
		AND (VINT.STATE_Off OR NOT CONF_VINT)
		 THEN
				OP_Arret_Pompes.Etape.3:=TRUE;
				OP_Arret_Pompes.Etape.2:=FALSE;
(*étape 3-4*)
ELSIF 	OP_Arret_Pompes.Etape.3
		AND	Timer_Arret_PP11.Q THEN 
				OP_Arret_Pompes.Etape.4:=TRUE;
				OP_Arret_Pompes.Etape.3:=FALSE;
(*étape 4-5*)
ELSIF	OP_Arret_Pompes.Etape.4
		AND PP11.STATE_Off AND PR11.STATE_Off AND PS11.STATE_Ar THEN
				OP_Arret_Pompes.Etape.5:=TRUE;
				OP_Arret_Pompes.Etape.4:=FALSE;
END_IF;

(*cloture du traitement de l'opération*)
OP_Arret_Pompes.POST();

(************************************************************************)
(*Gestion de la mémoire de la demande d'isolement de l'enceinte*)
(************************************************************************)
IF 		OP_Ventilation.Etape.9 THEN
	VAR_mem_isolement	:=	TRUE;
ELSIF	NOT OP_Pompage_Prim.AR OR NOT OP_Pompage_Sec.AR OR NOT OP_Pompage_Proc.AR OR NOT OP_Purge.AR THEN
	VAR_mem_isolement	:=	FALSE;
END_IF
(*IF OP_Arret_pompes.Etape.2 AND (NOT OP_Pompage_Prim.Etape.0  OR NOT OP_Pompage_Proc.Etape.0 OR NOT OP_Pompage_Sec.Etape.0) THEN
	VAR_mem_isolement_enceinte := TRUE;
END_IF;
IF OP_Arret_pompes.Etape.0 OR OP_Arret_Pompes.Etape.3 THEN
	VAR_mem_isolement_enceinte := FALSE;
END_IF;*)
END_ACTION

ACTION ACT_ISOLEMENT:
(*OPERATION ISOLEMENT ENCEINTE*)
(*isolement de l'enceinte*)

(*initialisation de l'opération*)
OP_Isolement(
	CTRL_PLC:= CTRL_PLC,
	RESET:= RESET,
	ENABLE_INT:=TRUE,
	MANUAL:= MANUAL,
	ON_AUTO_INT:= 	((DEF_TGF.DEF OR DEF_RP_enc.DEF) AND (NOT OP_Pompage_Prim.Etape.0 OR NOT OP_Pompage_Sec.Etape.0 OR NOT OP_Pompage_proc.Etape.0))
					OR (PS11.STATE_Nok AND (NOT OP_Pompage_Sec.Etape.0 OR NOT OP_Pompage_proc.Etape.0))
					OR (PP11.STATE_Nok AND NOT OP_Pompage_Prim.Etape.0)
					OR (PR11.STATE_NOK AND NOT OP_Pompage_Prim.Etape.0),
	RESTART_ENABLE_IF_OK:= FALSE,
	N_STEP_OP_OK:= 4,
	N_STEP_OP_NOK:=0);

(*appel de l'action de préparation de l'opération*)
OP_Isolement.PRL();


(*GRAFCET*)
(* initialisation du grafcet*)
IF 		OP_Isolement.Etape = 0
		THEN
				OP_Isolement.Etape.0	:= TRUE;
(*repositionnement sur étape 0*)
ELSIF	MANUAL OR RESET OR OP_pompage_sec.Etape.1 OR OP_Pompage_Proc.Etape.1 OR Op_Pompage_Prim.Etape.1
		OR OP_ventilation.Etape.2 OR OP_Ventilation.Etape.9 OR OP_Purge.Etape.1 THEN
				OP_Isolement.Etape := 0;
				OP_Isolement.Etape.0:=TRUE;
(*étape 0-1*)
ELSIF 	OP_Isolement.Etape.0
		AND(
		OP_Isolement.Marche_OP OR
		OP_ventilation.Etape.1 OR
		OP_Test_RP.Etape.3 OR
		(OP_Arret_Pompes.Etape.2 AND NOT VAR_mem_isolement) OR
		OP_Regen.Etape.2 OR OP_Regen_Part.Etape.2
		)
		THEN
				OP_Isolement.Etape.1:=TRUE;
				OP_Isolement.Etape.0:=FALSE;
(*étape 1-2*)
ELSIF	OP_Isolement.Etape.1
		AND OP_Pompage_Proc.Etape.0
		AND OP_Pompage_Prim.Etape.0
		AND OP_Pompage_Sec.Etape.0
		AND (OP_Ventilation.Etape.0 OR OP_Ventilation.Etape.1)
		AND (OP_Purge.Etape.0 OR (OP_Purge.Etape.4 AND OP_Ventilation.Etape.1))
		THEN
				OP_Isolement.Etape.2:=TRUE;
				OP_Isolement.Etape.1:=FALSE;
(*étape 2-3*)
ELSIF 	OP_Isolement.Etape.2 AND
		VP11.STATE_Off AND
		VS11.STATE_Off AND
		VH11.STATE_Off  THEN
				OP_Isolement.Etape.3:=TRUE;
				OP_Isolement.Etape.2:=FALSE;
(*étape 3-4*)
ELSIF	OP_Isolement.Etape.3
		AND ((PP11.STATE_Off AND PR11.STATE_Off) OR PS11.STATE_Regen OR CONF_Pompage_interjoint) THEN
				OP_isolement.Etape.4:=TRUE;
				OP_isolement.Etape.3:=FALSE;
END_IF;

(*cloture du traitement de l'opération*)
OP_Isolement.POST();
END_ACTION

ACTION ACT_MARCHE_POMPES:
(* OPERATION MARCHE POMPES*)
(* mise en marche des pompes*)

(*initialisation de l'opération*)
OP_MARCHE_POMPES(
	CTRL_PLC:= CTRL_PLC,
	RESET:= RESET,
	ENABLE_INT:=TRUE,
	MANUAL:= MANUAL,
	ON_AUTO_INT:= TRUE,
	RESTART_ENABLE_IF_OK:= FALSE,
	N_STEP_OP_OK:= 5,
	N_STEP_OP_NOK:=0);

(*appel de l'action de préparation de l'opération*)
OP_MARCHE_POMPES.PRL();


(*GRAFCET*)
(* initialisation du grafcet*)
IF 		OP_MARCHE_POMPES.ETAPE = 0
		THEN
				OP_MARCHE_POMPES.ETAPE.0 := TRUE;
(*repositionnement sur étape 0*)
ELSIF	MANUAL OR RESET OR OP_ARRET_POMPES.ETAPE.1
		THEN
				OP_MARCHE_POMPES.ETAPE := 0;			(*RAZ grafcet*)
				OP_MARCHE_POMPES.ETAPE.0:=TRUE;
(*étape 0-1*)
ELSIF 	OP_MARCHE_POMPES.ETAPE.0
		AND (OP_MARCHE_POMPES.MARCHE_OP OR OP_POMPAGE_SEC.ETAPE.2
			OR (OP_Regen.Etape.5 AND TH_Atm))
		THEN
				OP_MARCHE_POMPES.ETAPE.1:=TRUE;
				OP_MARCHE_POMPES.ETAPE.0:=FALSE;
(*étape 1-2*)
ELSIF	OP_MARCHE_POMPES.ETAPE.1
		AND OP_ARRET_POMPES.ETAPE.0 AND PR11.STATE_Off AND I_Ref_Ok
		THEN
				OP_MARCHE_POMPES.ETAPE.2:=TRUE;
				OP_MARCHE_POMPES.ETAPE.1:=FALSE;
(*étape 2-3*)
ELSIF 	OP_MARCHE_POMPES.ETAPE.2
		AND (PP11.STATE_On OR NOT CONF_Pompage_interjoint)
		THEN
				OP_MARCHE_POMPES.ETAPE.3:=TRUE;
				OP_MARCHE_POMPES.ETAPE.2:=FALSE;
(*étape 3-4*)
ELSIF	OP_MARCHE_POMPES.ETAPE.3
		THEN
				OP_MARCHE_POMPES.ETAPE.4:=TRUE;
				OP_MARCHE_POMPES.ETAPE.3:=FALSE;
(*étape 4-5*)
ELSIF 	OP_MARCHE_POMPES.ETAPE.4
		AND PS11.STATE_On AND PS11.STATE_Ok AND NOT PS11.STATE_Regen
		THEN
				OP_MARCHE_POMPES.ETAPE.5:=TRUE;
				OP_MARCHE_POMPES.ETAPE.4:=FALSE;
(*étape 5-4*)
ELSIF 	OP_MARCHE_POMPES.ETAPE.5
		AND (PS11.STATE_Regen OR NOT PS11.STATE_Ok)		THEN
				OP_MARCHE_POMPES.ETAPE.4:=TRUE;
				OP_MARCHE_POMPES.ETAPE.5:=FALSE;
END_IF;

(*cloture du traitement de l'opération*)
OP_MARCHE_POMPES.POST();
END_ACTION

ACTION ACT_POMPAGE_INTERJOINT:
(*GRAFCET*)
(* initialisation du grafcet*)
IF 		G7_pompage_interjoint.etape = 0
		THEN
				G7_pompage_interjoint.etape.0 := TRUE;
(*repositionnement sur étape 0*)
ELSIF	MANUAL OR RESET
		OR (NOT OP_POMPAGE_SEC.OK AND NOT OP_Pompage_Proc.OK AND NOT OP_Pompage_Proc.EC)
		OR NOT CONF_Pompage_interjoint OR NOT CONF_VINT
		THEN
				G7_pompage_interjoint.etape := 0;			(*RAZ grafcet*)
				G7_pompage_interjoint.etape.0:=TRUE;
(*étape 0-1*)
ELSIF 	G7_pompage_interjoint.etape.0
		AND (OP_POMPAGE_SEC.OK OR OP_Pompage_Proc.EC OR OP_Pompage_Proc.OK)
		THEN
				G7_pompage_interjoint.etape.1:=TRUE;
				G7_pompage_interjoint.etape.0:=FALSE;
(*étape 1-2*)
ELSIF	G7_pompage_interjoint.etape.1
		AND TIMER_pompage_interjoint.Q
		THEN
				G7_pompage_interjoint.etape.2:=TRUE;
				G7_pompage_interjoint.etape.1:=FALSE;
END_IF;

G7_pompage_interjoint.POST();
END_ACTION

ACTION ACT_POMPAGE_PRIM:
(*OPERATION POMPAGE PRIMAIRE ENCEINTE*)
(*pompage primaire dans l'enceinte*)

(*initialisation de l'opération*)
OP_POMPAGE_PRIM(
	CTRL_PLC:= CTRL_PLC,
	RESET:= RESET,
	ENABLE_INT:= OP_Purge.Etape.0 AND IN_FE11T AND IN_FE12T,
	MANUAL:= MANUAL,
	RESTART_ENABLE_IF_OK:= FALSE,
	N_STEP_OP_OK:= 5,
	N_STEP_OP_NOK:=0);

(*appel de l'action de préparation de l'opération*)
OP_POMPAGE_PRIM.PRL();


(*GRAFCET*)
(* initialisation du grafcet*)
IF 		OP_Pompage_Prim.Etape = 0
		THEN
				OP_Pompage_Prim.Etape.0:= TRUE;
(*repositionnement sur étape 0*)
ELSIF	MANUAL OR RESET OR OP_Isolement.Etape.1 OR OP_Pompage_Sec.Etape.4
		OR OP_Pompage_Proc.Etape.1
		THEN
				OP_Pompage_Prim.ETAPE := 0;
				OP_Pompage_Prim.Etape.0:=TRUE;
(*étape 0-1*)
ELSIF 	OP_Pompage_Prim.Etape.0
		AND (OP_Pompage_Prim.Marche_OP OR OP_Pompage_Sec.Etape.3 OR OP_Purge.Etape.2)
		THEN
				OP_Pompage_Prim.Etape.1:=TRUE;
				OP_Pompage_Prim.Etape.0:=FALSE;
(*étape 1-2*)
ELSIF	OP_Pompage_Prim.Etape.1
		AND OP_Isolement.Etape.0
		AND OP_Ventilation.Etape.0
		AND OP_Pompage_Proc.Etape.0
		AND (OP_Pompage_Sec.Etape.0 OR OP_Pompage_Sec.Etape.3)
		AND (OP_Purge.Etape.0 OR OP_Purge.Etape.6 OR OP_Purge.Etape.2)
		AND VS11.STATE_Off
		AND VH11.STATE_Off
		THEN
				OP_Pompage_Prim.Etape.2:=TRUE;
				OP_Pompage_Prim.Etape.1:=FALSE;

(*étape 2-3*)
ELSIF 	OP_Pompage_prim.Etape.2
		THEN
				OP_Pompage_Prim.Etape.3:=TRUE;
				OP_Pompage_Prim.Etape.2:=FALSE;
(*étape 3-4*)
ELSIF	OP_Pompage_Prim.Etape.3
		AND PP11.STATE_On AND PR11.STATE_On THEN
				OP_Pompage_Prim.Etape.4:=TRUE;
				OP_Pompage_Prim.Etape.3:=FALSE;
(*étape 4-5*)
ELSIF 	OP_Pompage_Prim.Etape.4
		AND VP11.STATE_On
		THEN
				OP_Pompage_Prim.Etape.5:=TRUE;
				OP_Pompage_Prim.Etape.4:=FALSE;
END_IF;

(*cloture du traitement de l'opération*)
OP_Pompage_Prim.POST();
END_ACTION

ACTION ACT_POMPAGE_PROC:
(*OPERATION POMPAGE PROCEDE*)
(*pompage procede dans l'enceinte*)

(*initialisation de l'opération*)
OP_Pompage_Proc(
	CTRL_PLC:= CTRL_PLC,
	RESET:= RESET,
	ENABLE_INT:= OP_POMPAGE_SEC.OK OR OP_Pompage_Proc.OK,
	MANUAL:= MANUAL,
	RESTART_ENABLE_IF_OK:= FALSE,
	N_STEP_OP_OK:= 3,
	N_STEP_OP_NOK:=0);

(*appel de l'action de préparation de l'opération*)
OP_Pompage_Proc.PRL();


(*GRAFCET*)
(* initialisation du grafcet*)
IF 		OP_Pompage_Proc.Etape = 0
		THEN
				OP_Pompage_Proc.Etape.0:= TRUE;
(*repositionnement sur étape 0*)
ELSIF	MANUAL OR RESET OR OP_Isolement.Etape.1 OR OP_Pompage_Prim.Etape.1 OR OP_Pompage_Sec.Etape.1
		OR OP_Purge.Etape.1
		THEN
				OP_Pompage_Proc.Etape := 0;
				OP_Pompage_Proc.Etape.0:=TRUE;
(*étape 0-1*)
ELSIF 	OP_Pompage_Proc.Etape.0
		AND OP_Pompage_Proc.Marche_OP
		THEN
				OP_Pompage_Proc.Etape.1:=TRUE;
				OP_Pompage_Proc.Etape.0:=FALSE;
(*étape 1-2*)
ELSIF	OP_Pompage_Proc.Etape.1
		AND OP_Pompage_Sec.Etape.0
		THEN
				OP_Pompage_Proc.Etape.2:=TRUE;
				OP_Pompage_Proc.Etape.1:=FALSE;
(*étape 2-3*)
ELSIF 	OP_Pompage_proc.Etape.2
		AND VS11.STATE_Lam THEN
				OP_Pompage_Proc.Etape.3:=TRUE;
				OP_Pompage_Proc.Etape.2:=FALSE;
(*étape 3-2*)
ELSIF 	OP_Pompage_Proc.Etape.3
		AND OP_Pompage_Proc.Marche_OP
		THEN
				OP_Pompage_Proc.Etape.2:=TRUE;
				OP_Pompage_Proc.Etape.3:=FALSE;
END_IF;

(*cloture du traitement de l'opération*)
OP_Pompage_Proc.POST();
END_ACTION

ACTION ACT_POMPAGE_SEC:
(*OPERATION POMPAGE SECONDAIRE ENCEINTE*)
(*pompage secondaire dans l'enceinte*)

(*initialisation de l'opération*)
OP_pompage_sec(
	CTRL_PLC:= CTRL_PLC,
	RESET:= RESET,
	ENABLE_INT:=IN_FE11T AND IN_FE12T AND NOT PS11.STATE_Regen,
	MANUAL:= MANUAL,
	RESTART_ENABLE_IF_OK:= FALSE,
	N_STEP_OP_OK:= 7,
	N_STEP_OP_NOK:=0);

(*appel de l'action de préparation de l'opération*)
OP_Pompage_Sec.PRL();


(*GRAFCET*)
(* initialisation du grafcet*)
IF 		OP_Pompage_Sec.Etape = 0
		THEN
				OP_Pompage_Sec.Etape.0:= TRUE;
(*repositionnement sur étape 0*)
ELSIF	MANUAL OR RESET OR OP_Isolement.Etape.1 OR OP_Pompage_Proc.Etape.1
		OR (OP_Pompage_Prim.Etape.1 AND NOT OP_Pompage_Sec.Etape.3) OR OP_Purge.Etape.1
		THEN
				OP_Pompage_Sec.Etape := 0;
				OP_Pompage_Sec.Etape.0:=TRUE;
(*étape 0-1*)
ELSIF 	OP_Pompage_Sec.Etape.0 AND
		(OP_Pompage_Sec.Marche_OP OR OP_Purge.Etape.6 OR
			OP_Test_RP.Etape.2 OR OP_Test_RP.Etape.7
		OR (OP_Regen.Etape.5 AND NOT TH_Atm AND OP_Pompage_Sec.ENABLE_INT))
		THEN
				OP_Pompage_Sec.Etape.1:=TRUE;
				OP_Pompage_Sec.Etape.0:=FALSE;
(*étape 1-2*)
ELSIF	OP_Pompage_Sec.Etape.1
		AND OP_Isolement.Etape.0
		AND OP_Ventilation.Etape.0
		AND OP_Pompage_Proc.Etape.0
		AND (OP_Purge.Etape.0 OR OP_Purge.Etape.6)
		THEN
				OP_Pompage_Sec.Etape.2:=TRUE;
				OP_Pompage_Sec.Etape.1:=FALSE;
(*étape 2-3*)
ELSIF 	OP_Pompage_Sec.Etape.2
		AND OP_MARCHE_POMPES.ok AND NOT TH_Vide_Primaire AND VH11.STATE_Off
		THEN
				OP_Pompage_Sec.Etape.3:=TRUE;
				OP_Pompage_Sec.Etape.2:=FALSE;
(*étape 2-4*)
ELSIF 	OP_Pompage_Sec.Etape.2
		AND OP_MARCHE_POMPES.ok AND TH_Vide_Primaire AND VH11.STATE_Off
		THEN
				OP_Pompage_Sec.Etape.4:=TRUE;
				OP_Pompage_Sec.Etape.2:=FALSE;
(*étape 3-4*)
ELSIF	OP_Pompage_Sec.Etape.3
		AND	OP_POMPAGE_PRIM.ok  AND TH_Vide_Primaire
		THEN
				OP_Pompage_Sec.Etape.4:=TRUE;
				OP_Pompage_Sec.Etape.3:=FALSE;
(*étape 4-5*)
ELSIF	OP_Pompage_Sec.Etape.4
		AND VP11.STATE_Off
		AND  OP_POMPAGE_PRIM.AR   THEN
				OP_Pompage_Sec.Etape.5:=TRUE;
				OP_Pompage_Sec.Etape.4:=FALSE;
(*étape 5-6*)
ELSIF 	OP_Pompage_Sec.Etape.5
		AND (PP11.STATE_Off AND PR11.STATE_Off OR CONF_Pompage_interjoint)
		THEN
				OP_Pompage_Sec.Etape.6:=TRUE;
				OP_Pompage_Sec.Etape.5:=FALSE;
(*étape 6-7*)
ELSIF 	OP_Pompage_Sec.Etape.6
		AND VS11.STATE_On
		THEN
				OP_Pompage_Sec.Etape.7:=TRUE;
				OP_Pompage_Sec.Etape.6:=FALSE;
END_IF;

(*cloture du traitement de l'opération*)
OP_Pompage_Sec.POST();
END_ACTION

ACTION ACT_PURGE:
(*OPERATION PURGE*)
(*purge enceinte : pompage primaire pendant un temps donné puis ventilation, répété X fois*)

(*initialisation de l'opération*)
OP_Purge(
	CTRL_PLC:= CTRL_PLC,
	RESET:= RESET,
	ENABLE_INT:= IN_FE11T AND IN_FE12T AND OP_Test_RP.AR,
	MANUAL:= MANUAL,
	RESTART_ENABLE_IF_OK:= FALSE,
	N_STEP_OP_OK:= 7,
	N_STEP_OP_NOK:=0);

(*appel de l'action de préparation de l'opération*)
OP_Purge.PRL();


(*GRAFCET*)
(* initialisation du grafcet*)
IF 		OP_Purge.Etape = 0
		THEN
				OP_Purge.Etape.0:= TRUE;
(*repositionnement sur étape 0*)
ELSIF	MANUAL OR RESET OR OP_Arret_Pompes.Etape.1
		OR (OP_Isolement.Etape.1 AND NOT OP_Ventilation.Etape.1)
		OR (OP_Pompage_Sec.Etape.1 AND NOT OP_Purge.Etape.6)
		THEN
				OP_Purge.Etape := 0;
				OP_Purge.Etape.0:=TRUE;
(*étape 0-1*)
ELSIF 	OP_Purge.Etape.0
		AND OP_Purge.Marche_OP
		THEN
				OP_Purge.Etape.1:=TRUE;
				OP_Purge.Etape.0:=FALSE;
(*étape 1-2*)
ELSIF	OP_Purge.Etape.1
		AND OP_Pompage_Sec.Etape.0 AND OP_Pompage_Prim.Etape.0 AND OP_Pompage_Proc.Etape.0
		AND OP_Ventilation.Etape.0 AND OP_Isolement.Etape.0
		THEN
				OP_Purge.Etape.2:=TRUE;
				OP_Purge.Etape.1:=FALSE;
(*étape 2-3*)
ELSIF 	OP_Purge.Etape.2
		AND OP_Pompage_Prim.OK AND TH_Vide_Primaire
		THEN
				OP_Purge.Etape.3:=TRUE;
				OP_Purge.Etape.2:=FALSE;
(*étape 3-4*)
ELSIF 	OP_Purge.Etape.3
		AND TIMER_Purge.Q
		THEN
				OP_Purge.Etape.4:=TRUE;
				OP_Purge.Etape.3:=FALSE;
(*étape 3-2*)
ELSIF 	OP_Purge.Etape.3
		AND NOT OP_Pompage_Prim.OK
		THEN
				OP_Purge.Etape.2:=TRUE;
				OP_Purge.Etape.3:=FALSE;
(*étape 4-5*)
ELSIF 	OP_Purge.Etape.4
		AND TH_Atm
		THEN
				OP_Purge.Etape.5:=TRUE;
				OP_Purge.Etape.4:=FALSE;
(*étape 5-2*)
ELSIF 	OP_Purge.Etape.5
		AND (VAR_Iter_Purge < PRM_N_Purge)
		THEN
				OP_Purge.Etape.2:=TRUE;
				OP_Purge.Etape.5:=FALSE;
(*étape 5-6*)
ELSIF 	OP_Purge.Etape.5
		AND (VAR_Iter_Purge >= PRM_N_Purge)
		THEN
				OP_Purge.Etape.6:=TRUE;
				OP_Purge.Etape.5:=FALSE;
(*étape 6-7*)
ELSIF 	OP_Purge.Etape.6
		AND OP_Pompage_Sec.EC
		THEN
				OP_Purge.Etape.7:=TRUE;
				OP_Purge.Etape.6:=FALSE;
END_IF;

(*cloture du traitement de l'opération*)
OP_Purge.POST();
END_ACTION

ACTION ACT_REGEN:
(*OPERATION REGENERATION POMPE CRYOGENIQUE*)
(*isolement pompage et lancement régénération*)

(*initialisation de l'opération*)
OP_Regen(
	CTRL_PLC:= CTRL_PLC,
	RESET:= RESET,
	ENABLE_INT:= OP_Test_RP.AR AND NOT OP_Marche_Pompes.AR,
	MANUAL:= MANUAL,
	RESTART_ENABLE_IF_OK:= FALSE,
	N_STEP_OP_OK:= 6,
	N_STEP_OP_NOK:=0);

(*appel de l'action de préparation de l'opération*)
OP_Regen.PRL();


(*GRAFCET*)
(* initialisation du grafcet*)
IF 		OP_Regen.Etape = 0
		THEN
				OP_Regen.Etape.0:= TRUE;
(*repositionnement sur étape 0*)
ELSIF	MANUAL OR RESET OR OP_Arret_Pompes.Etape.1
		THEN
				OP_Regen.Etape := 0;
				OP_Regen.Etape.0:=TRUE;
(*étape 0-1*)
ELSIF 	OP_Regen.Etape.0
		AND (OP_Regen.Marche_OP OR (FM_REGEN.Q AND NOT MANUAL AND NOT OP_Regen_Part.EC))
		THEN
				OP_Regen.Etape.1:=TRUE;
				OP_Regen.Etape.0:=FALSE;
(*étape 1-2*)
ELSIF	OP_Regen.Etape.1
		THEN
				OP_Regen.Etape.2:=TRUE;
				OP_Regen.Etape.1:=FALSE;
(*étape 2-3*)
ELSIF 	OP_Regen.Etape.2
		AND (OP_Isolement.Etape.4 OR (OP_Pompage_Prim.Etape.0 AND OP_Pompage_Proc.Etape.0 OR OP_Pompage_Sec.Etape.0 OR OP_Purge.Etape.0))
		THEN
				OP_Regen.Etape.3:=TRUE;
				OP_Regen.Etape.2:=FALSE;
(*étape 3-4*)
ELSIF	OP_Regen.Etape.3 AND PS11.STATE_Regen
		THEN
				OP_Regen.Etape.4:=TRUE;
				OP_Regen.Etape.3:=FALSE;
(*étape 4-5*)
ELSIF	OP_Regen.Etape.4 AND NOT PS11.STATE_Regen
		THEN
				OP_Regen.Etape.5:=TRUE;
				OP_Regen.Etape.4:=FALSE;
(*étape 5-6*)
ELSIF	OP_Regen.Etape.5
		AND (OP_Pompage_Sec.OK OR (OP_Marche_Pompes.OK AND (TH_Atm OR NOT OP_Pompage_Sec.ENABLE_INT)))
		THEN
				OP_Regen.Etape.6:=TRUE;
				OP_Regen.Etape.5:=FALSE;
(*étape 6-0*)
ELSIF	OP_Regen.Etape.6
		AND TIMER_etape6_regen.Q
		THEN
				OP_Regen.Etape.0:=TRUE;
				OP_Regen.Etape.6:=FALSE;
END_IF;

(*cloture du traitement de l'opération*)
OP_Regen.POST();
END_ACTION

ACTION ACT_REGEN_PART:
(*OPERATION REGENERATION POMPE CRYOGENIQUE*)
(*isolement pompage et lancement régénération*)

(*initialisation de l'opération*)
OP_Regen_Part(
	CTRL_PLC:= CTRL_PLC,
	RESET:= RESET,
	ENABLE_INT:= OP_Test_RP.AR AND NOT OP_Marche_Pompes.AR,
	MANUAL:= MANUAL,
	RESTART_ENABLE_IF_OK:= FALSE,
	N_STEP_OP_OK:= 6,
	N_STEP_OP_NOK:=0);

(*appel de l'action de préparation de l'opération*)
OP_Regen_Part.PRL();


(*GRAFCET*)
(* initialisation du grafcet*)
IF 		OP_Regen_Part.Etape = 0
		THEN
				OP_Regen_Part.Etape.0:= TRUE;
(*repositionnement sur étape 0*)
ELSIF	MANUAL OR RESET OR OP_Arret_Pompes.Etape.1
		OR OP_Pompage_Sec.Etape.1 OR OP_Pompage_Prim.Etape.1
		THEN
				OP_Regen_Part.Etape := 0;
				OP_Regen_Part.Etape.0:=TRUE;
(*étape 0-1*)
ELSIF 	OP_Regen_Part.Etape.0
		AND OP_Regen_Part.Marche_OP
		THEN
				OP_Regen_Part.Etape.1:=TRUE;
				OP_Regen_Part.Etape.0:=FALSE;
(*étape 1-2*)
ELSIF	OP_Regen_Part.Etape.1
		THEN
				OP_Regen_Part.Etape.2:=TRUE;
				OP_Regen_Part.Etape.1:=FALSE;
(*étape 2-3*)
ELSIF 	OP_Regen_Part.Etape.2
		AND (OP_Isolement.OK
		OR (OP_Pompage_Prim.Etape.0 AND OP_Pompage_Proc.Etape.0 OR OP_Pompage_Sec.Etape.0 OR OP_Purge.Etape.0))
		THEN
				OP_Regen_Part.Etape.3:=TRUE;
				OP_Regen_Part.Etape.2:=FALSE;
(*étape 3-4*)
ELSIF	OP_Regen_Part.Etape.3 AND PS11.STATE_Regen
		THEN
				OP_Regen_Part.Etape.4:=TRUE;
				OP_Regen_Part.Etape.3:=FALSE;
(*étape 4-5*)
ELSIF	OP_Regen_Part.Etape.4
		AND IN_Temp_Etage1 > 300
		THEN
				OP_Regen_Part.Etape.5:=TRUE;
				OP_Regen_Part.Etape.4:=FALSE;
(*étape 5-6*)
ELSIF	OP_Regen_Part.Etape.5
		AND (IN_Temp_Etage1 < PRM_Temp_Post_Purge
			OR TIMER_Post_Purge.Q )
		THEN
				OP_Regen_Part.Etape.6:=TRUE;
				OP_Regen_Part.Etape.5:=FALSE;
(*étape 6-0*)
ELSIF	OP_Regen_Part.Etape.6
		AND TIMER_etape6_regen.Q
		THEN
				OP_Regen_Part.Etape.0:=TRUE;
				OP_Regen_Part.Etape.6:=FALSE;
END_IF;

(*cloture du traitement de l'opération*)
OP_Regen_Part.POST();
END_ACTION

ACTION ACT_TEST_RP:
(*OPERATION TEST REMONTEE PRESSION*)

OP_TEST_RP(
	CTRL_PLC:= CTRL_PLC,
	RESET:= RESET,
	MANUAL:=MANUAL ,
	ENABLE_INT := OP_Pompage_Sec.OK AND OP_Purge.AR AND OP_Regen.AR AND OP_Regen_Part.AR,
	RESTART_ENABLE_IF_OK:=TRUE ,
	N_STEP_OP_OK:= 8,
	N_STEP_OP_NOK:=0 );

(*appel de l'action de préparation de l'opération*)
OP_TEST_RP.PRL();

(*GRAFCET*)
(* initialisation du grafcet*)
IF 		OP_TEST_RP.ETAPE = 0
		THEN
				OP_TEST_RP.ETAPE.0 := TRUE;
(*repositionnement sur étape 0*)
ELSIF 	RESET OR MANUAL OR (OP_Isolement.Etape.1 AND NOT OP_Test_RP.Etape.3)
			OR (OP_Pompage_Sec.Etape.1 AND OP_Test_RP.Etape.3) OR CO_Stop_Test_RP
			OR OP_Arret_Pompes.Etape.1 OR OP_Isolement.ON_AUTO_EXT OR OP_Isolement.ON_AUTO_INT
		THEN
				OP_TEST_RP.ETAPE := 0;
				OP_TEST_RP.ETAPE.0:=TRUE;
(*étape 0-1*)
ELSIF 	OP_TEST_RP.ETAPE.0 AND OP_TEST_RP.MARCHE_OP
		THEN
				OP_TEST_RP.ETAPE.1:=TRUE;
				OP_TEST_RP.ETAPE.0:=FALSE;
(*étape 1-2*)
ELSIF 	OP_TEST_RP.ETAPE.1
		THEN
				OP_TEST_RP.ETAPE.2:=TRUE;
				OP_TEST_RP.ETAPE.1:=FALSE;
(*étape 2-3*)
ELSIF 	OP_TEST_RP.ETAPE.2
		AND OP_Pompage_Sec.ok AND TH_Test_RP
		THEN
				OP_TEST_RP.ETAPE.3:=TRUE;
				OP_TEST_RP.ETAPE.2:=FALSE;
(*étape 3-4*)
ELSIF 	OP_TEST_RP.ETAPE.3
		AND OP_Isolement.OK
		THEN
				OP_TEST_RP.ETAPE.4:=TRUE;
				OP_TEST_RP.ETAPE.3:=FALSE;
(*étape 4-5*)
ELSIF 	OP_TEST_RP.ETAPE.4
		AND TIMER_attente_test.Q
		THEN
				OP_TEST_RP.ETAPE.5:=TRUE;
				OP_TEST_RP.ETAPE.4:=FALSE;
(*étape 5-6*)
ELSIF 	OP_TEST_RP.ETAPE.5
		THEN
				OP_TEST_RP.ETAPE.6:=TRUE;
				OP_TEST_RP.ETAPE.5:=FALSE;
(*étape 6-7*)
ELSIF 	OP_TEST_RP.ETAPE.6
		THEN
				OP_TEST_RP.ETAPE.7:=TRUE;
				OP_TEST_RP.ETAPE.6:=FALSE;
(*étape 7-8*)
ELSIF 	OP_TEST_RP.ETAPE.7
		AND OP_Pompage_Sec.OK
		THEN
				OP_TEST_RP.ETAPE.8:=TRUE;
				OP_TEST_RP.ETAPE.7:=FALSE;
(*étape 8-1*)
ELSIF 	OP_TEST_RP.ETAPE.8 AND OP_TEST_RP.MARCHE_OP
		THEN
				OP_TEST_RP.ETAPE.1:=TRUE;
				OP_TEST_RP.ETAPE.8:=FALSE;
END_IF
(*cloture du traitement de l'opération*)
OP_TEST_RP.POST();
CO_Stop_Test_RP	:=	FALSE;
END_ACTION

ACTION ACT_VENTILATION:
(*OPERATION VENTILATION*)


(*initialisation de l'opération*)
OP_Ventilation(
	CTRL_PLC:= CTRL_PLC,
	RESET:= RESET,
	ENABLE_INT:=OP_Purge.Etape.0,
	MANUAL:= MANUAL,
	ON_AUTO_INT:= FALSE ,
	RESTART_ENABLE_IF_OK:= FALSE,
	N_STEP_OP_OK:= 8,
	N_STEP_OP_NOK:=0);

(*appel de l'action de préparation de l'opération*)
OP_Ventilation.PRL();


(*GRAFCET*)
(* initialisation du grafcet*)
IF 		OP_Ventilation.Etape = 0
		THEN
				OP_Ventilation.Etape.0:= TRUE;
(*repositionnement sur étape 0*)
ELSIF	MANUAL OR RESET OR (OP_isolement.Etape.1 AND NOT  OP_ventilation.Etape.1)
		OR OP_Pompage_sec.Etape.1 OR Op_Pompage_Prim.Etape.1
		OR OP_Pompage_Proc.Etape.1 OR OP_Purge.Etape.1
		THEN
				OP_Ventilation.Etape := 0;
				OP_Ventilation.Etape.0:=TRUE;
(*étape 0-1*)
ELSIF 	OP_Ventilation.Etape.0
		 AND (OP_Ventilation.Marche_OP OR OP_Purge.Etape.4)
		THEN
				OP_Ventilation.Etape.1:=TRUE;
				OP_Ventilation.Etape.0:=FALSE;
(*étape 1-9*)
ELSIF	OP_Ventilation.Etape.1
		AND OP_isolement.OK THEN
				OP_Ventilation.Etape.9:=TRUE;
				OP_Ventilation.Etape.1:=FALSE;
(*étape 9-2*)
ELSIF	OP_Ventilation.Etape.9
		AND OP_isolement.Etape.0 THEN
				OP_Ventilation.Etape.2:=TRUE;
				OP_Ventilation.Etape.9:=FALSE;
(*étape 2-3*)
ELSIF 	OP_Ventilation.Etape.2 AND  I_Prep_Ventil_Ok  THEN
				OP_Ventilation.Etape.3:=TRUE;
				OP_Ventilation.Etape.2:=FALSE;
(*étape 3-4*)
ELSIF	OP_Ventilation.Etape.3
		AND  I_Stop_Mesure_OK   THEN
				OP_Ventilation.Etape.4:=TRUE;
				OP_Ventilation.Etape.3:=FALSE;
(*étape 4-5*)
ELSIF	OP_Ventilation.Etape.4
		THEN
				OP_Ventilation.Etape.5:=TRUE;
				OP_Ventilation.Etape.4:=FALSE;
(*étape 5-6*)
ELSIF 	OP_Ventilation.Etape.5
		AND (TH_atm OR I_Fin_Ventil OR NOT IN_FE11T OR NOT IN_FE12T )
		THEN
				OP_Ventilation.Etape.6:=TRUE;
				OP_Ventilation.Etape.5:=FALSE;
(*étape 6-7*)
ELSIF 	OP_Ventilation.Etape.6
		AND (TIMER_SurVentilation_enc.Q OR I_Fin_Ventil OR NOT IN_FE11T OR NOT IN_FE12T)
		THEN
				OP_Ventilation.Etape.7:=TRUE;
				OP_Ventilation.Etape.6:=FALSE;
(*étape 7-8*)
ELSIF 	OP_Ventilation.Etape.7
		AND VH11.STATE_Off THEN
				OP_Ventilation.Etape.8:=TRUE;
				OP_Ventilation.Etape.7:=FALSE;
END_IF;

(*cloture du traitement de l'opération*)
OP_Ventilation.POST();
END_ACTION

ACTION POST:
VAR_Reset_Sortie := 	NOT MANUAL AND OP_Arret_Pompes.Etape.0 AND OP_Isolement.Etape.0 AND OP_Marche_Pompes.Etape.0
					AND OP_Pompage_Prim.Etape.0 AND OP_Pompage_Proc.Etape.0 AND OP_Pompage_Sec.Etape.0
					AND OP_Ventilation.Etape.0 AND OP_Purge.Etape.0 AND OP_Regen.Etape.0 AND OP_Regen_Part.Etape.0;




(*****************************************)
(*       pompe primaire PP11             *)
(*****************************************)
IF (OP_MARCHE_POMPES.ETAPE.2 AND CONF_Pompage_interjoint)
	OR OP_Pompage_Prim.Etape.3
	OR PS11.STATE_Regen AND NOT RESET
	THEN
		PP11.CO_On 	:= 	TRUE;
ELSIF RESET OR (VAR_Reset_Sortie AND NOT PS11.STATE_Regen)
    OR (OP_Pompage_Sec.Etape.5 AND PR11.STATE_Off AND NOT CONF_Pompage_interjoint)
	OR (OP_Isolement.Etape.3 AND PR11.STATE_Off AND NOT PS11.STATE_Regen  AND NOT CONF_Pompage_interjoint)
	OR OP_Arret_Pompes.Etape.4 AND PR11.STATE_Off AND VP11.STATE_Off
	THEN
		PP11.CO_On	:= 	FALSE;
END_IF;

(*****************************************)
(*       pompe primaire PR11             *)
(*****************************************)
TIMER_Arret_Roots.IN := (OP_Pompage_Sec.OK
						OR (OP_Pompage_Prim.AR AND VP11.STATE_Off AND NOT PS11.STATE_Regen)) AND CONF_Pompage_interjoint;
TIMER_Arret_Roots.PT := T#2M;

TIMER_Arret_Roots();

IF (OP_Pompage_Prim.Etape.3 AND PP11.STATE_On)
	OR (PS11.STATE_Regen AND PP11.STATE_On AND NOT RESET) THEN
		PR11.CO_On 	:= 	TRUE;
ELSIF RESET OR VAR_Reset_Sortie
    OR TIMER_Arret_Roots.Q
	OR OP_Arret_Pompes.Etape.3 
	OR (OP_Isolement.Etape.3 AND NOT PS11.STATE_Regen AND NOT CONF_Pompage_interjoint)
	OR (OP_Pompage_Sec.Etape.5 AND NOT CONF_Pompage_interjoint)
	THEN
		PR11.CO_On	:= 	FALSE;
END_IF;

(*****************************************)
(* 		pompe cryo PS11		   *)
(*****************************************)
IF  OP_Marche_Pompes.Etape.4  THEN
	PS11.CO_On 	:= 	TRUE;
ELSIF RESET  (*OR VAR_Reset_Sortie TODOLN*)  OR OP_Arret_Pompes.Etape.3 THEN
	PS11.CO_On	:= 	FALSE;
	PS11.CO_Regen := FALSE;
END_IF;
IF OP_Regen.Etape.3 OR OP_Regen_Part.Etape.3 THEN
	PS11.CO_Regen	:=	TRUE;
ELSIF OP_Regen.Etape.4 OR OP_Regen_Part.Etape.4 THEN
	PS11.CO_Regen	:=	FALSE;
ELSIF MANUAL THEN
	PS11.CO_On		:=	PS11.VAR_On;
END_IF;

(*****************************************)
(* 		vanne VP11    		   *)
(*****************************************)
IF OP_Pompage_Prim.Etape.4   THEN
		VP11.CO_On 		:= 	TRUE;
ELSIF RESET OR VAR_Reset_Sortie OR OP_Pompage_Sec.Etape.4  OR OP_Isolement.Etape.2 THEN
		VP11.CO_On		:= 	FALSE;
END_IF;


(******************************************)
(*		Vanne  VH11		              *)
(******************************************)
IF   OP_VENTILATION.Etape.5 OR OP_Ventilation.Etape.6 THEN
			VH11.CO_On 	:= 	TRUE;
ELSIF RESET OR  VAR_Reset_Sortie OR OP_Pompage_Prim.Etape.1 OR
	   OP_Pompage_Sec.Etape.2 OR   OP_Isolement.Etape.2 OR OP_Ventilation.Etape.7
	   THEN
			VH11.CO_On	:= 	FALSE;
END_IF;

(******************************************)
(*                  Vanne  VS11                       *)
(******************************************)
IF OP_Pompage_Sec.Etape.6   THEN
		VS11.CO_On 	:= 	TRUE;
		VS11.CO_Lam:=	FALSE;
ELSIF OP_Pompage_Proc.Etape.2  THEN
		VS11.CO_On 	:= 	FALSE;
		VS11.CO_Lam:=	TRUE;
ELSIF VAR_Reset_Sortie OR RESET
	   OR OP_Pompage_Prim.Etape.1   OR OP_Isolement.Etape.2 THEN
		VS11.CO_On	:= 	FALSE;
		VS11.CO_Lam:=	FALSE;
END_IF;


(******************************************)
(*                 Vanne  VINT                        *)
(******************************************)
IF G7_pompage_interjoint.etape.2  THEN
		VINT.CO_On 	:= 	TRUE;
ELSIF VAR_Reset_Sortie OR RESET OR (G7_pompage_interjoint.etape.0 AND NOT MANUAL)
	THEN
		VINT.CO_On	:= 	FALSE;
END_IF;



(***********************************************)
(*                Demande diverse              *)
(***********************************************)

(*demande de préparation avant ventilation*)
RQ_Prep_Ventil_Enc 	:= OP_VENTILATION.Etape.2;

(*Demande d'arrêt de la mesure avant ventilation enceinte*)
RQ_Stop_Mesure_Enc := Op_Ventilation.Etape.3 OR Op_Ventilation.Etape.4 OR Op_Ventilation.Etape.5 ;

(*Tempo de surventilation enceinte*)
TIMER_SurVentilation_Enc	(
					PT:=PRM_Tim_SurVentil_E,
					IN:=OP_VENTILATION.Etape.6 AND TH_Atm
					);

(*Temporisation d'arrêt pompe primaire*)
TIMER_Arret_PP11(
					PT:=PRM_Tim_Arret_PP11,
					IN:=OP_Arret_Pompes.Etape.3,
				);

(*Tempo de purge*)
TIMER_Purge (
					PT:=PRM_Tim_Purge,
					IN:=OP_Purge.Etape.3
					);

(*Compteur d'itération purge*)
IF		OP_Purge.Etape.0 THEN
	VAR_Iter_Purge	:=	0;
ELSIF	OP_Purge.Etape.5 THEN
	VAR_Iter_Purge	:=	VAR_Iter_Purge + 1;
END_IF

(*timer de prep ventil*)
TIM_Prep_ventil.PT := PRM_Tim_Prep_Ventil;
TIM_Prep_ventil.IN := OP_Ventilation.Etape.2;
TIM_Prep_ventil();


(*Tempo de retard à l'ouverture de la vanne interjoint*)
TIMER_pompage_interjoint(
					PT:=T#30s,
					IN:=G7_pompage_interjoint.etape.1
					);


(*timer de post purge en regen partielle*)
TIMER_Post_Purge.PT			:=	PRM_Tim_Post_Purge;
TIMER_Post_Purge.IN			:=	OP_Regen_Part.Etape.5;
TIMER_Post_Purge();

TIMER_etape6_regen.PT		:=	T#500ms;
TIMER_etape6_regen.IN		:=	OP_Regen.Etape.6 OR OP_Regen_Part.Etape.6;
TIMER_etape6_regen();

(***************** test de remontée de pression*************************)
TIMER_attente_test		(
					PT:=PRM_Tim_test,
					IN:=OP_Test_RP.Etape.4
					);
(*Mémorisation des pressions lors du test et calcul de l'indicateur*)
IF FM_etape4.Q THEN
	VAR_Mem_Pression_deb := IN_Pressure_RP;
END_IF;
IF OP_Test_RP.Etape.5 THEN
	VAR_Mem_Pression_fin := IN_Pressure_RP;
END_IF;
(*Indicateur final faisant intervenir le volume ATTENTION : FORMULE MEMO SANS DOUTE FAUSSE*)
IF OP_Test_RP.Etape.6 THEN
	VAR_indicateur_test := (VAR_Mem_Pression_fin - VAR_Mem_Pression_deb) * CONF_volume_enceinte / TIME_TO_REAL(PRM_Tim_Test) * 1000;
END_IF;



(*****************************************************)
(* APPEL DES FONCTIONS COMPOSANTS*)
(*****************************************************)

(*Vanne de pompage primaire enceinte*)
VP11(
	RESET:= RESET,
	MANUAL:= MANUAL,
	EN_On_INT:=  PP11.STATE_On AND PR11.STATE_On AND VH11.STATE_Off AND VS11.STATE_Off AND IN_FE11T AND IN_FE12T AND NOT PS11.STATE_Regen,
	EN_Off_INT:= TRUE
	);

(*Vanne pompage secondaire enceinte*)
VS11(
	RESET:= RESET,
	MANUAL:= MANUAL,
	EN_On_INT:= (PS11.STATE_Ok
				AND VP11.STATE_Off AND VH11.STATE_Off)
				AND TH_RP_Enc,
	EN_Off_INT:= TRUE
	);

(*Vanne ventilation enceinte*)
VH11(
	RESET:= RESET,
	MANUAL:= MANUAL,
	EN_On_INT:= VP11.STATE_Off  AND  VS11.STATE_Off,
	EN_Off_INT:= TRUE
	);

(*Vanne interjoint*)
VINT(
	RESET:= RESET,
	MANUAL:= MANUAL,
	EN_On_INT:= PP11.STATE_On AND NOT PS11.STATE_Regen,
	EN_Off_INT:= TRUE
	);

(*Pompe primaire PP11*)
PP11(
	RESET:= 	RESET,
	MANUAL:= 	MANUAL AND NOT PS11.STATE_Regen,
	EN_On_INT:= TRUE,
	EN_Off_INT:= (PR11.STATE_Off AND VP11.STATE_Off AND NOT PS11.STATE_Regen) OR VAR_Reset_sortie
	);
	
(*Pompe roots PR11*)
PR11(
	RESET:= 	RESET,
	MANUAL:= 	MANUAL,
	EN_On_INT:= PP11.STATE_On,
	EN_Off_INT:= (VP11.STATE_Off AND NOT PS11.STATE_Regen) OR VAR_Reset_sortie
	);

(*Pompe cryo PS11*)
PS11(
	RESET:= RESET,
	MANUAL:= MANUAL,
	EN_On_INT:= TRUE ,
	EN_Off_INT:= VS11.STATE_Off OR VAR_Reset_Sortie,
	EN_Regen_INT:= VS11.STATE_Off
	);


(*******************************************)
(* GESTION DES DEFAUTS 	     *)
(*******************************************)


(*Défaut d'obtention du seuil de basculement en pompage secondaire*)
DEF_PPRIM			(
					Condition:=	(OP_Pompage_Prim.Etape.5 AND OP_Pompage_Sec.Etape.3) AND (DEF_PPRIM.DELAY<>T#0ms)

					);
DEF_TGF				(
					Condition:= 	(OP_Pompage_Prim.Etape.5 OR OP_pompage_prim.Etape.4) AND OP_Pompage_sec.Etape.3
								AND	(DEF_TGF.DELAY<>T#0ms) AND NOT TH_Grosse_Fuite
					);

(*Défaut de remontée de pression dans l'enceinte pendant le pompage secondaire*)
(* validation ok - SP *)
DEF_RP_enc			(
					Condition:=	NOT VS11.STATE_Off AND NOT TH_RP_Enc AND NOT RESET
					);

(*Défaut de ventilation*)
DEF_Vent			(
					Condition:=	(OP_ventilation.Etape.4 OR Op_ventilation.Etape.5 OR op_ventilation.Etape.6) AND (DEF_Vent.DELAY <> T#0ms)
					);
END_ACTION

ACTION PRL:
(*vérification pour empécher la division par 0*)
IF TIME_TO_REAL(PRM_Tim_test) = 0 THEN
	PRM_Tim_test := T#1s;
END_IF
FM_etape4(clk := OP_Test_RP.Etape.4);

	IdXML							:=	'2';
	TagXML							:=	0;

	OP_Marche_Pompes.IdXML			:= 	'1';
	OP_Marche_Pompes.TagXML			:=	1;

	OP_Arret_Pompes.IdXML			:= 	'1';
	OP_Arret_Pompes.TagXML			:= 	2;

	OP_Isolement.IdXML				:= 	'1';
	OP_Isolement.TagXML				:= 	3;

	OP_Ventilation.IdXML			:= 	'1';
	OP_Ventilation.TagXML			:= 	4;

	OP_Pompage_Prim.IdXML			:=	'1';
	OP_Pompage_Prim.TagXML			:=	6;

	OP_Pompage_Sec.IdXML			:=	'1';
	OP_Pompage_Sec.TagXML			:=	5;

	OP_Pompage_Proc.IdXML			:=	'1';
	OP_Pompage_Proc.TagXML			:=	7;

	OP_Purge.IdXML					:=	'1';
	OP_Purge.TagXML					:=	8;

	OP_Regen.IdXML					:=	'1';
	OP_Regen.TagXML					:=	9;

	OP_Test_RP.IdXML				:=	'1';
	OP_Test_RP.TagXML				:=	10;


	DEF_PPrim.IdXML			:= '1';
	DEF_PPrim.TagXML		:= 1;
	DEF_Vent.IdXML			:= '1';
	DEF_Vent.TagXML			:= 2;
	DEF_RP_enc.IdXML		:= '1';
	DEF_RP_enc.TagXML		:= 3;
	DEF_TGF.IdXML			:= '1';
	DEF_TGF.TagXML			:= 4;

	PP11.IdXML					:=	'1';
	PP11.TagXML					:=	7;
	
	PR11.IdXML					:=	'1';
	PR11.TagXML					:=	10;

	PS11.IdXML					:=	'1';
	PS11.TagXML					:=	9;

	VP11.IdXML					:=	'1';
	VP11.TagXML					:=	2;
	VP11.DEF_On.IdXML			:=	'3';
	VP11.DEF_On.TagXML			:=	2;
	VP11.DEF_Off.IdXML			:=	'3';
	VP11.DEF_Off.TagXML			:=	4;
	VP11.DEF_Sensor.IdXML		:=	'3';
	VP11.DEF_Sensor.TagXML		:=	13;
	VP11.DEF_On_Imposs.IdXML	:=	'3';
	VP11.DEF_On_Imposs.TagXML	:=	6;
	VP11.DEF_Off_Imposs.IdXML	:=	'3';
	VP11.DEF_Off_Imposs.TagXML	:=	9;
	VP11.DEF_Off_auto.IdXML		:=	'3';
	VP11.DEF_Off_auto.TagXML	:=	11;

